      ;FOLD F328 = AUS ;%{SE}%MKUKATPVW %CVW_SPS %VBOASG %P 2:F328 = AUS, 3: BOASG
         $FLAG[328] = FALSE
      ;ENDFOLD
      ;FOLD F324 = AUS ;%{SE}%MKUKATPVW %CVW_SPS %VBOASG %P 2:F324 = AUS, 3: BOASG
         $FLAG[324] = FALSE
      ;ENDFOLD
      ;FOLD Schritt 151 = A4039 ;%{SE}%MKUKATPVW %CVW_SPS %VST_CON %P 2:Schritt 151 = A4039, 3: ST_CON
         IF $OUT[4039] THEN
            PREV_STEP[9] = APP_INT_STEP[9]
            APP_INT_STEP[9] = 151
         ENDIF
      ;ENDFOLD
   ;ENDFOLD
   ;FOLD SCHRITT 151 -- st. RZ1 # Fehler Fraesen -- ;%{P}%MKUKATPVW,%CSTEP,%VST_NR,%P 1:SCHRITT, 2:151, 3: st. RZ1 # Fehler Fraesen
      ;FOLD ;%{H}
         Case 151
      ;ENDFOLD
      ;FOLD -- Fehler Reset AUS -- ;%{SE}%MKUKATPVW %CVW_COM %VCOMMENT %P 2:-- Fehler Reset AUS --, 3: VW_COMMENT
      ;ENDFOLD
      ;FOLD A3857 = AUS ;%{SE}%MKUKATPVW %CVW_SPS %VBOASG %P 2:A3857 = AUS, 3: BOASG
         $OUT[3857] = FALSE
      ;ENDFOLD
      ;FOLD -- Start StartAcknowledge EIN -- ;%{SE}%MKUKATPVW %CVW_COM %VCOMMENT %P 2:-- Start StartAcknowledge EIN --, 3: VW_COMMENT
      ;ENDFOLD
      ;FOLD A3512 = EIN ;%{SE}%MKUKATPVW %CVW_SPS %VBOASG %P 2:A3512 = EIN, 3: BOASG
         $OUT[3512] = TRUE
      ;ENDFOLD
      ;FOLD Schritt 152 = A4039 ;%{SE}%MKUKATPVW %CVW_SPS %VST_CON %P 2:Schritt 152 = A4039, 3: ST_CON
         IF $OUT[4039] THEN
            PREV_STEP[9] = APP_INT_STEP[9]
            APP_INT_STEP[9] = 152
         ENDIF
      ;ENDFOLD
   ;ENDFOLD
   ;FOLD SCHRITT 152 -- st. RZ1 # Fehler Fraesen -- ;%{P}%MKUKATPVW,%CSTEP,%VST_NR,%P 1:SCHRITT, 2:152, 3: st. RZ1 # Fehler Fraesen
      ;FOLD ;%{H}
         Case 152
      ;ENDFOLD
      ;FOLD -- Start StartAcknowledge AUS -- ;%{SE}%MKUKATPVW %CVW_COM %VCOMMENT %P 2:-- Start StartAcknowledge AUS --, 3: VW_COMMENT
      ;ENDFOLD
      ;FOLD A3512 = AUS ;%{SE}%MKUKATPVW %CVW_SPS %VBOASG %P 2:A3512 = AUS, 3: BOASG
         $OUT[3512] = FALSE
      ;ENDFOLD
      ;FOLD -- Start Dress in Position AUS -- ;%{SE}%MKUKATPVW %CVW_COM %VCOMMENT %P 2:-- Start Dress in Position AUS --, 3: VW_COMMENT
      ;ENDFOLD
      ;FOLD A3871 = AUS ;%{SE}%MKUKATPVW %CVW_SPS %VBOASG %P 2:A3871 = AUS, 3: BOASG
         $OUT[3871] = FALSE
      ;ENDFOLD
      ;FOLD -- Start Dress Fin AUS -- ;%{SE}%MKUKATPVW %CVW_COM %VCOMMENT %P 2:-- Start Dress Fin AUS --, 3: VW_COMMENT
      ;ENDFOLD
      ;FOLD A3872 = AUS ;%{SE}%MKUKATPVW %CVW_SPS %VBOASG %P 2:A3872 = AUS, 3: BOASG
         $OUT[3872] = FALSE
      ;ENDFOLD
      ;FOLD -- Start Dress AUS -- ;%{SE}%MKUKATPVW %CVW_COM %VCOMMENT %P 2:-- Start Dress AUS --, 3: VW_COMMENT
      ;ENDFOLD
      ;FOLD A3510 = EIN ;%{SE}%MKUKATPVW %CVW_SPS %VBOASG %P 2:A3510 = EIN, 3: BOASG
         $OUT[3510] = TRUE
      ;ENDFOLD
      ;FOLD -- Start Spot AUS -- ;%{SE}%MKUKATPVW %CVW_COM %VCOMMENT %P 2:-- Start Spot AUS --, 3: VW_COMMENT
      ;ENDFOLD
      ;FOLD A3511 = AUS ;%{SE}%MKUKATPVW %CVW_SPS %VBOASG %P 2:A3511 = AUS, 3: BOASG
         $OUT[3511] = FALSE
      ;ENDFOLD
      ;FOLD -- Start Spot AUS -- ;%{SE}%MKUKATPVW %CVW_COM %VCOMMENT %P 2:-- Start Spot AUS --, 3: VW_COMMENT
      ;ENDFOLD
      ;FOLD A3511 = AUS ;%{SE}%MKUKATPVW %CVW_SPS %VBOASG %P 2:A3511 = AUS, 3: BOASG
         $OUT[3511] = FALSE
      ;ENDFOLD
      ;FOLD -- Start Init Same AUS -- ;%{SE}%MKUKATPVW %CVW_COM %VCOMMENT %P 2:-- Start Init Same AUS --, 3: VW_COMMENT
      ;ENDFOLD
      ;FOLD A3514 = AUS ;%{SE}%MKUKATPVW %CVW_SPS %VBOASG %P 2:A3514 = AUS, 3: BOASG
         $OUT[3514] = FALSE
      ;ENDFOLD
      ;FOLD -- Start Init New AUS -- ;%{SE}%MKUKATPVW %CVW_COM %VCOMMENT %P 2:-- Start Init New AUS --, 3: VW_COMMENT
      ;ENDFOLD
      ;FOLD A3513 = AUS ;%{SE}%MKUKATPVW %CVW_SPS %VBOASG %P 2:A3513 = AUS, 3: BOASG
         $OUT[3513] = FALSE
      ;ENDFOLD
      ;FOLD A3518 = A3519 ;%{SE}%MKUKATPVW %CVW_SPS %VBOASG %P 2:A3518 = A3519, 3: BOASG
         $OUT[3518] = $OUT[3519]
      ;ENDFOLD
      ;FOLD Schritt 153 = A4039 & A3862 ;%{SE}%MKUKATPVW %CVW_SPS %VST_CON %P 2:Schritt 153 = A4039 & A3862, 3: ST_CON
         IF $OUT[4039] AND $OUT[3862] THEN
            PREV_STEP[9] = APP_INT_STEP[9]
            APP_INT_STEP[9] = 153
         ENDIF
      ;ENDFOLD
   ;ENDFOLD
   ;FOLD SCHRITT 153 -- st. RZ1 # Fehler Fraesen -- ;%{P}%MKUKATPVW,%CSTEP,%VST_NR,%P 1:SCHRITT, 2:153, 3: st. RZ1 # Fehler Fraesen
      ;FOLD ;%{H}
         Case 153
      ;ENDFOLD
      ;FOLD -- RSK Fehlerausgabe KF Versetzeinheit -- ;%{SE}%MKUKATPVW %CVW_COM %VCOMMENT %P 2:-- RSK Fehlerausgabe KF Versetzeinheit --, 3: VW_COMMENT
      ;ENDFOLD
      ;FOLD F328 = E835 & F564 ;%{SE}%MKUKATPVW %CVW_SPS %VBOASG %P 2:F328 = E835 & F564, 3: BOASG
         $FLAG[328] = $IN[835] AND $FLAG[564]
      ;ENDFOLD
      ;FOLD -- RSK Fehlerausgabe KS1 Arbeitsstellung -- ;%{SE}%MKUKATPVW %CVW_COM %VCOMMENT %P 2:-- RSK Fehlerausgabe KS1 Arbeitsstellung --, 3: VW_COMMENT
      ;ENDFOLD
      ;FOLD F324 = (E836 + !E837 + !E838 + E839) ;%{SE}%MKUKATPVW %CVW_SPS %VBOASG %P 2:F324 = (E836 + !E837 + !E838 + E839), 3: BOASG
         $FLAG[324] = ($IN[836] OR NOT $IN[837] OR NOT $IN[838] OR $IN[839])
      ;ENDFOLD
      ;FOLD A3519 = EIN ;%{SE}%MKUKATPVW %CVW_SPS %VBOASG %P 2:A3519 = EIN, 3: BOASG
         $OUT[3519] = TRUE
      ;ENDFOLD
      ;FOLD Schritt 154 = A4039 & A3862 & A3505 & A3506 & !A3518 & (E26 + E27) ;%{SE}%MKUKATPVW %CVW_SPS %VST_CON %P 2:Schritt 154 = A4039 & A3862 & A3505 & A3506 & !A3518 & (E26 + E27), 3: ST_CON
         IF $OUT[4039] AND $OUT[3862] AND $OUT[3505] AND $OUT[3506] AND NOT $OUT[3518] AND ($IN[26] OR $IN[27]) THEN
            PREV_STEP[9] = APP_INT_STEP[9]
            APP_INT_STEP[9] = 154
         ENDIF
      ;ENDFOLD
      ;FOLD Schritt 116 = A4039 & A3862 & A3505 & A3506 & A3518 & (E26 + E27) ;%{SE}%MKUKATPVW %CVW_SPS %VST_CON %P 2:Schritt 116 = A4039 & A3862 & A3505 & A3506 & A3518 & (E26 + E27), 3: ST_CON
         IF $OUT[4039] AND $OUT[3862] AND $OUT[3505] AND $OUT[3506] AND $OUT[3518] AND ($IN[26] OR $IN[27]) THEN
            PREV_STEP[9] = APP_INT_STEP[9]
            APP_INT_STEP[9] = 116
         ENDIF
      ;ENDFOLD
   ;ENDFOLD
   ;FOLD SCHRITT 154 -- st. RZ1 # Fehler Fraesen -- ;%{P}%MKUKATPVW,%CSTEP,%VST_NR,%P 1:SCHRITT, 2:154, 3: st. RZ1 # Fehler Fraesen
      ;FOLD ;%{H}
         Case 154
      ;ENDFOLD
      ;FOLD -- Fehler ruecksetzen -- ;%{SE}%MKUKATPVW %CVW_COM %VCOMMENT %P 2:-- Fehler ruecksetzen --, 3: VW_COMMENT
      ;ENDFOLD
      ;FOLD A140 = AUS ;%{SE}%MKUKATPVW %CVW_SPS %VBOASG %P 2:A140 = AUS, 3: BOASG
         $OUT[140] = FALSE
      ;ENDFOLD
      ;FOLD A144 = AUS ;%{SE}%MKUKATPVW %CVW_SPS %VBOASG %P 2:A144 = AUS, 3: BOASG
         $OUT[144] = FALSE
      ;ENDFOLD
      ;FOLD Schritt 103 = (F324 + F328) & E836 & !E837 & !E838 & E839 & A4039 ;%{SE}%MKUKATPVW %CVW_SPS %VST_CON %P 2:Schritt 103 = (F324 + F328) & E836 & !E837 & !E838 & E839 & A4039, 3: ST_CON
         IF ($FLAG[324] OR $FLAG[328]) AND $IN[836] AND NOT $IN[837] AND NOT $IN[838] AND $IN[839] AND $OUT[4039] THEN
            PREV_STEP[9] = APP_INT_STEP[9]
            APP_INT_STEP[9] = 103
         ENDIF
      ;ENDFOLD
      ;FOLD SCHRITT 111 = !F324 & !F328 & !E836 & E837 & E838 & !E839 & A4039 ;%{SE}%MKUKATPVW %CVW_SPS %VST_CON %P 2:SCHRITT 111 = !F324 & !F328 & !E836 & E837 & E838 & !E839 & A4039, 3: ST_CON
         IF NOT $FLAG[324] AND NOT $FLAG[328] AND NOT $IN[836] AND $IN[837] AND $IN[838] AND NOT $IN[839] AND $OUT[4039] THEN
            PREV_STEP[9] = APP_INT_STEP[9]
            APP_INT_STEP[9] = 111
         ENDIF
      ;ENDFOLD
   ;ENDFOLD
   ;FOLD SCHRITT 155 -- st. RZ1 # Fehler Fraesen  -- ;%{P}%MKUKATPVW,%CSTEP,%VST_NR,%P 1:SCHRITT, 2:155, 3: st. RZ1 # Fehler Fraesen
      ;FOLD ;%{H}
         Case 155
      ;ENDFOLD
      ;FOLD Schritt 111 = A4039 & A3506 & A3505 ;%{SE}%MKUKATPVW %CVW_SPS %VST_CON %P 2:Schritt 111 = A4039 & A3506 & A3505, 3: ST_CON
         IF $OUT[4039] AND $OUT[3506] AND $OUT[3505] THEN
            PREV_STEP[9] = APP_INT_STEP[9]
            APP_INT_STEP[9] = 111
         ENDIF
      ;ENDFOLD
   ;ENDFOLD
   ;FOLD SCHRITT 160 -- st. RZ1 # Fehler Messen -- ;%{P}%MKUKATPVW,%CSTEP,%VST_NR,%P 1:SCHRITT, 2:160, 3: st. RZ1 # Fehler Messen
      ;FOLD ;%{H}
         Case 160
      ;ENDFOLD
      ;FOLD 1:;%{SE} %MKUKATPVW
      ;ENDFOLD
   ;ENDFOLD
   ;FOLD SCHRITT 161 -- st. RZ1 # Fehler Messen -- ;%{P}%MKUKATPVW,%CSTEP,%VST_NR,%P 1:SCHRITT, 2:161, 3: st. RZ1 # Fehler Messen
      ;FOLD ;%{H}
         Case 161
      ;ENDFOLD
      ;FOLD -- Fehler Reset AUS -- ;%{SE}%MKUKATPVW %CVW_COM %VCOMMENT %P 2:-- Fehler Reset AUS --, 3: VW_COMMENT
      ;ENDFOLD
      ;FOLD A3857 = AUS ;%{SE}%MKUKATPVW %CVW_SPS %VBOASG %P 2:A3857 = AUS, 3: BOASG
         $OUT[3857] = FALSE
      ;ENDFOLD
      ;FOLD -- Anwahl Zange 1 EIN -- ;%{SE}%MKUKATPVW %CVW_COM %VCOMMENT %P 2:-- Anwahl Zange 1 EIN --, 3: VW_COMMENT
      ;ENDFOLD
      ;FOLD A3858 = EIN ;%{SE}%MKUKATPVW %CVW_SPS %VBOASG %P 2:A3858 = EIN, 3: BOASG
         $OUT[3858] = TRUE
      ;ENDFOLD
      ;FOLD -- Start StartAcknowledge EIN -- ;%{SE}%MKUKATPVW %CVW_COM %VCOMMENT %P 2:-- Start StartAcknowledge EIN --, 3: VW_COMMENT
      ;ENDFOLD
      ;FOLD A3512 = EIN ;%{SE}%MKUKATPVW %CVW_SPS %VBOASG %P 2:A3512 = EIN, 3: BOASG
         $OUT[3512] = TRUE
      ;ENDFOLD
      ;FOLD Schritt 162 = A4039 & A140 & A3862 ;%{SE}%MKUKATPVW %CVW_SPS %VST_CON %P 2:Schritt 162 = A4039 & A140 & A3862, 3: ST_CON
         IF $OUT[4039] AND $OUT[140] AND $OUT[3862] THEN
            PREV_STEP[9] = APP_INT_STEP[9]
            APP_INT_STEP[9] = 162
         ENDIF
      ;ENDFOLD
   ;ENDFOLD
   ;FOLD SCHRITT 162 -- st. RZ1 # Fehler Messen -- ;%{P}%MKUKATPVW,%CSTEP,%VST_NR,%P 1:SCHRITT, 2:162, 3: st. RZ1 # Fehler Messen
      ;FOLD ;%{H}
         Case 162
      ;ENDFOLD
      ;FOLD -- Start Init Same AUS -- ;%{SE}%MKUKATPVW %CVW_COM %VCOMMENT %P 2:-- Start Init Same AUS --, 3: VW_COMMENT
      ;ENDFOLD
      ;FOLD A3514 = AUS ;%{SE}%MKUKATPVW %CVW_SPS %VBOASG %P 2:A3514 = AUS, 3: BOASG
         $OUT[3514] = FALSE
      ;ENDFOLD
      ;FOLD -- Start Spot AUS -- ;%{SE}%MKUKATPVW %CVW_COM %VCOMMENT %P 2:-- Start Spot AUS --, 3: VW_COMMENT
      ;ENDFOLD
      ;FOLD A3511 = AUS ;%{SE}%MKUKATPVW %CVW_SPS %VBOASG %P 2:A3511 = AUS, 3: BOASG
         $OUT[3511] = FALSE
      ;ENDFOLD
      ;FOLD -- Start Dress AUS -- ;%{SE}%MKUKATPVW %CVW_COM %VCOMMENT %P 2:-- Start Dress AUS --, 3: VW_COMMENT
      ;ENDFOLD
      ;FOLD A3510 = AUS ;%{SE}%MKUKATPVW %CVW_SPS %VBOASG %P 2:A3510 = AUS, 3: BOASG
         $OUT[3510] = FALSE
      ;ENDFOLD
      ;FOLD -- Start Init New AUS -- ;%{SE}%MKUKATPVW %CVW_COM %VCOMMENT %P 2:-- Start Init New AUS --, 3: VW_COMMENT
      ;ENDFOLD
      ;FOLD A3513 = AUS ;%{SE}%MKUKATPVW %CVW_SPS %VBOASG %P 2:A3513 = AUS, 3: BOASG
         $OUT[3513] = FALSE
      ;ENDFOLD
      ;FOLD -- Start Dress in Position AUS -- ;%{SE}%MKUKATPVW %CVW_COM %VCOMMENT %P 2:-- Start Dress in Position AUS --, 3: VW_COMMENT
      ;ENDFOLD
      ;FOLD A3871 = AUS ;%{SE}%MKUKATPVW %CVW_SPS %VBOASG %P 2:A3871 = AUS, 3: BOASG
         $OUT[3871] = FALSE
      ;ENDFOLD
      ;FOLD -- Start Dress Fin AUS -- ;%{SE}%MKUKATPVW %CVW_COM %VCOMMENT %P 2:-- Start Dress Fin AUS --, 3: VW_COMMENT
      ;ENDFOLD
      ;FOLD A3872 = AUS ;%{SE}%MKUKATPVW %CVW_SPS %VBOASG %P 2:A3872 = AUS, 3: BOASG
         $OUT[3872] = FALSE
      ;ENDFOLD
      ;FOLD -- Start StartAcknowledge AUS -- ;%{SE}%MKUKATPVW %CVW_COM %VCOMMENT %P 2:-- Start StartAcknowledge AUS --, 3: VW_COMMENT
      ;ENDFOLD
      ;FOLD A3512 = AUS ;%{SE}%MKUKATPVW %CVW_SPS %VBOASG %P 2:A3512 = AUS, 3: BOASG
         $OUT[3512] = FALSE
      ;ENDFOLD
      ;FOLD Schritt 163 = A4039 ;%{SE}%MKUKATPVW %CVW_SPS %VST_CON %P 2:Schritt 163 = A4039, 3: ST_CON
         IF $OUT[4039] THEN
            PREV_STEP[9] = APP_INT_STEP[9]
            APP_INT_STEP[9] = 163
         ENDIF
      ;ENDFOLD
   ;ENDFOLD
   ;FOLD SCHRITT 163 -- st. RZ1 # Fehler Messen -- ;%{P}%MKUKATPVW,%CSTEP,%VST_NR,%P 1:SCHRITT, 2:163, 3: st. RZ1 # Fehler Messen
      ;FOLD ;%{H}
         Case 163
      ;ENDFOLD
      ;FOLD Schritt 164 = A4039 & !A3507 & A3506 & (E26 + E27) ;%{SE}%MKUKATPVW %CVW_SPS %VST_CON %P 2:Schritt 164 = A4039 & !A3507 & A3506 & (E26 + E27), 3: ST_CON
         IF $OUT[4039] AND NOT $OUT[3507] AND $OUT[3506] AND ($IN[26] OR $IN[27]) THEN
            PREV_STEP[9] = APP_INT_STEP[9]
            APP_INT_STEP[9] = 164
         ENDIF
      ;ENDFOLD
   ;ENDFOLD
   ;FOLD SCHRITT 164 -- st. RZ1 # Fehler Messen -- ;%{P}%MKUKATPVW,%CSTEP,%VST_NR,%P 1:SCHRITT, 2:164, 3: st. RZ1 # Fehler Messen
      ;FOLD ;%{H}
         Case 164
      ;ENDFOLD
      ;FOLD Schritt 124 = A4039 & A140 & !A3507 & A3506 & A3505 & F959 ;%{SE}%MKUKATPVW %CVW_SPS %VST_CON %P 2:Schritt 124 = A4039 & A140 & !A3507 & A3506 & A3505 & F959, 3: ST_CON
         IF $OUT[4039] AND $OUT[140] AND NOT $OUT[3507] AND $OUT[3506] AND $OUT[3505] AND $FLAG[959] THEN
            PREV_STEP[9] = APP_INT_STEP[9]
            APP_INT_STEP[9] = 124
         ENDIF
      ;ENDFOLD
   ;ENDFOLD
   ;FOLD SCHRITT 165 --st.RZ1 # Fehler Schweissen-- ;%{P}%MKUKATPVW,%CSTEP,%VST_NR,%P 1:SCHRITT, 2:165, 3:st.RZ1 # Fehler Schweissen
      ;FOLD ;%{H}
         Case 165
      ;ENDFOLD
      ;FOLD -- Start StartAcknowledge AUS -- ;%{SE}%MKUKATPVW %CVW_COM %VCOMMENT %P 2:-- Start StartAcknowledge AUS --, 3: VW_COMMENT
      ;ENDFOLD
      ;FOLD A3512 = AUS ;%{SE}%MKUKATPVW %CVW_SPS %VBOASG %P 2:A3512 = AUS, 3: BOASG
         $OUT[3512] = FALSE
      ;ENDFOLD
      ;FOLD -- Start Dress in Position AUS -- ;%{SE}%MKUKATPVW %CVW_COM %VCOMMENT %P 2:-- Start Dress in Position AUS --, 3: VW_COMMENT
      ;ENDFOLD
      ;FOLD A3871 = AUS ;%{SE}%MKUKATPVW %CVW_SPS %VBOASG %P 2:A3871 = AUS, 3: BOASG
         $OUT[3871] = FALSE
      ;ENDFOLD
      ;FOLD -- Start Dress Fin AUS -- ;%{SE}%MKUKATPVW %CVW_COM %VCOMMENT %P 2:-- Start Dress Fin AUS --, 3: VW_COMMENT
      ;ENDFOLD
      ;FOLD A3872 = AUS ;%{SE}%MKUKATPVW %CVW_SPS %VBOASG %P 2:A3872 = AUS, 3: BOASG
         $OUT[3872] = FALSE
      ;ENDFOLD
      ;FOLD -- Start Dress AUS -- ;%{SE}%MKUKATPVW %CVW_COM %VCOMMENT %P 2:-- Start Dress AUS --, 3: VW_COMMENT
      ;ENDFOLD
      ;FOLD A3510 = AUS ;%{SE}%MKUKATPVW %CVW_SPS %VBOASG %P 2:A3510 = AUS, 3: BOASG
         $OUT[3510] = FALSE
      ;ENDFOLD
      ;FOLD -- Start Spot AUS -- ;%{SE}%MKUKATPVW %CVW_COM %VCOMMENT %P 2:-- Start Spot AUS --, 3: VW_COMMENT
      ;ENDFOLD
      ;FOLD A3511 = AUS ;%{SE}%MKUKATPVW %CVW_SPS %VBOASG %P 2:A3511 = AUS, 3: BOASG
         $OUT[3511] = FALSE
      ;ENDFOLD
      ;FOLD -- Start Spot AUS -- ;%{SE}%MKUKATPVW %CVW_COM %VCOMMENT %P 2:-- Start Spot AUS --, 3: VW_COMMENT
      ;ENDFOLD
      ;FOLD A3511 = AUS ;%{SE}%MKUKATPVW %CVW_SPS %VBOASG %P 2:A3511 = AUS, 3: BOASG
         $OUT[3511] = FALSE
      ;ENDFOLD
      ;FOLD -- Start Init Same AUS -- ;%{SE}%MKUKATPVW %CVW_COM %VCOMMENT %P 2:-- Start Init Same AUS --, 3: VW_COMMENT
      ;ENDFOLD
      ;FOLD A3514 = AUS ;%{SE}%MKUKATPVW %CVW_SPS %VBOASG %P 2:A3514 = AUS, 3: BOASG
         $OUT[3514] = FALSE
      ;ENDFOLD
      ;FOLD -- Start Init New AUS -- ;%{SE}%MKUKATPVW %CVW_COM %VCOMMENT %P 2:-- Start Init New AUS --, 3: VW_COMMENT
      ;ENDFOLD
      ;FOLD A3513 = AUS ;%{SE}%MKUKATPVW %CVW_SPS %VBOASG %P 2:A3513 = AUS, 3: BOASG
         $OUT[3513] = FALSE
      ;ENDFOLD
      ;FOLD A3533 = EIN ;%{SE}%MKUKATPVW %CVW_SPS %VBOASG %P 2:A3533 = EIN, 3: BOASG
         $OUT[3533] = TRUE
      ;ENDFOLD
      ;FOLD A130 = AUS ;%{SE}%MKUKATPVW %CVW_SPS %VBOASG %P 2:A130 = AUS, 3: BOASG
         $OUT[130] = FALSE
      ;ENDFOLD
      ;FOLD F92 = AUS ;%{SE}%MKUKATPVW %CVW_SPS %VBOASG %P 2:F92 = AUS, 3: BOASG
         $FLAG[92] = FALSE
      ;ENDFOLD
      ;FOLD Schritt 2 = A4039 & A3862 & A3506 & A3505 & (E26 + E27) ;%{SE}%MKUKATPVW %CVW_SPS %VST_CON %P 2:Schritt 2 = A4039 & A3862 & A3506 & A3505 & (E26 + E27), 3: ST_CON
         IF $OUT[4039] AND $OUT[3862] AND $OUT[3506] AND $OUT[3505] AND ($IN[26] OR $IN[27]) THEN
            PREV_STEP[9] = APP_INT_STEP[9]
            APP_INT_STEP[9] = 2
         ENDIF
      ;ENDFOLD
   ;ENDFOLD
   ;FOLD SCHRITT 166 --st.RZ1 # Fehler Schweissen-- ;%{P}%MKUKATPVW,%CSTEP,%VST_NR,%P 1:SCHRITT, 2:166, 3:st.RZ1 # Fehler Schweissen
      ;FOLD ;%{H}
         Case 166
      ;ENDFOLD
      ;FOLD 1:;%{SE} %MKUKATPVW
      ;ENDFOLD
   ;ENDFOLD
   ;FOLD SCHRITT 190 -- st. RZ1 Setzhub 2 -- ;%{P}%MKUKATPVW,%CSTEP,%VST_NR,%P 1:SCHRITT, 2:190, 3: st. RZ1 Setzhub 2
      ;FOLD ;%{H}
         Case 190
      ;ENDFOLD
      ;FOLD -- Druckvorgabe SK1/ServoGun -- ;%{SE}%MKUKATPVW %CVW_COM %VCOMMENT %P 2:-- Druckvorgabe SK1/ServoGun --, 3: VW_COMMENT
      ;ENDFOLD
      ;FOLD bin1 ( F78 ) = 61 ;%{SE}%MKUKATPVW %CVW_SPS %VARIASG %P 2:bin1 ( F78 ) = 61, 3: ARIASG
         VW(#BINOUT,$FLAG[78],1,61)
      ;ENDFOLD
      ;FOLD bin31 ( F78 ) = 61 ;%{SE}%MKUKATPVW %CVW_SPS %VARIASG %P 2:bin31 ( F78 ) = 61, 3: ARIASG
         VW(#BINOUT,$FLAG[78],31,61)
      ;ENDFOLD
      ;FOLD -- Wartezeit Programmwechsel SK -- ;%{SE}%MKUKATPVW %CVW_COM %VCOMMENT %P 2:-- Wartezeit Programmwechsel SK --, 3: VW_COMMENT
      ;ENDFOLD
      ;FOLD T8 ( !F334 ) = -2[1/10Sek] ;%{SE}%MKUKATPVW %CVW_SPS %VTASG %P 2:T8 ( !F334 ) = -2[1/10Sek], 3: TASG
         VW(#SET_TIME,NOT $FLAG[334],8,0,-2)
      ;ENDFOLD
      ;FOLD -- Ueberwachungszeit ServoGun Setzhub 2 -- ;%{SE}%MKUKATPVW %CVW_COM %VCOMMENT %P 2:-- Ueberwachungszeit ServoGun Setzhub 2 --, 3: VW_COMMENT
      ;ENDFOLD
      ;FOLD t9 ( EIN ) = -80[1/10Sek] ;%{SE}%MKUKATPVW %CVW_SPS %VTASG %P 2:t9 ( EIN ) = -80[1/10Sek], 3: TASG
         VW(#SET_TIME,TRUE,9,0,-80)
      ;ENDFOLD
      ;FOLD -- Hilfsflag SK Programmwechsel -- ;%{SE}%MKUKATPVW %CVW_COM %VCOMMENT %P 2:-- Hilfsflag SK Programmwechsel --, 3: VW_COMMENT
      ;ENDFOLD
      ;FOLD F334 = EIN ;%{SE}%MKUKATPVW %CVW_SPS %VBOASG %P 2:F334 = EIN, 3: BOASG
         $FLAG[334] = TRUE
      ;ENDFOLD
      ;FOLD A3512 = AUS ;%{SE}%MKUKATPVW %CVW_SPS %VBOASG %P 2:A3512 = AUS, 3: BOASG
         $OUT[3512] = FALSE
      ;ENDFOLD
      ;FOLD SCHRITT 191 = T8 & A4039 & A3506 & A3505 & !A3507 ;%{SE}%MKUKATPVW %CVW_SPS %VST_CON %P 2:SCHRITT 191 = T8 & A4039 & A3506 & A3505 & !A3507, 3: ST_CON
         IF $TIMER_FLAG[8] AND $OUT[4039] AND $OUT[3506] AND $OUT[3505] AND NOT $OUT[3507] THEN
            PREV_STEP[9] = APP_INT_STEP[9]
            APP_INT_STEP[9] = 191
         ENDIF
      ;ENDFOLD
   ;ENDFOLD
   ;FOLD SCHRITT 191 -- st. RZ1 Setzhub 2 # InitSame -- ;%{P}%MKUKATPVW,%CSTEP,%VST_NR,%P 1:SCHRITT, 2:191, 3: st. RZ1 Setzhub 2 # InitSame
      ;FOLD ;%{H}
         Case 191
      ;ENDFOLD
      ;FOLD -- Hilfsflag SK Programmwechsel -- ;%{SE}%MKUKATPVW %CVW_COM %VCOMMENT %P 2:-- Hilfsflag SK Programmwechsel --, 3: VW_COMMENT
      ;ENDFOLD
      ;FOLD F334 = AUS ;%{SE}%MKUKATPVW %CVW_SPS %VBOASG %P 2:F334 = AUS, 3: BOASG
         $FLAG[334] = FALSE
      ;ENDFOLD
      ;FOLD -- Zeit fuer Setzhub -- ;%{SE}%MKUKATPVW %CVW_COM %VCOMMENT %P 2:-- Zeit fuer Setzhub --, 3: VW_COMMENT
      ;ENDFOLD
      ;FOLD T8 ( EIN ) = -80[1/10Sek] ;%{SE}%MKUKATPVW %CVW_SPS %VTASG %P 2:T8 ( EIN ) = -80[1/10Sek], 3: TASG
         VW(#SET_TIME,TRUE,8,0,-80)
      ;ENDFOLD
      ;FOLD -- Messen nach Fraesen -- ;%{SE}%MKUKATPVW %CVW_COM %VCOMMENT %P 2:-- Messen nach Fraesen --, 3: VW_COMMENT
      ;ENDFOLD
      ;FOLD A3514 = EIN ;%{SE}%MKUKATPVW %CVW_SPS %VBOASG %P 2:A3514 = EIN, 3: BOASG
         $OUT[3514] = TRUE
      ;ENDFOLD
      ;FOLD A3510 = EIN ;%{SE}%MKUKATPVW %CVW_SPS %VBOASG %P 2:A3510 = EIN, 3: BOASG
         $OUT[3510] = TRUE
      ;ENDFOLD
      ;FOLD SCHRITT 192 = A4039 ;%{SE}%MKUKATPVW %CVW_SPS %VST_CON %P 2:SCHRITT 192 = A4039, 3: ST_CON
         IF $OUT[4039] THEN
            PREV_STEP[9] = APP_INT_STEP[9]
            APP_INT_STEP[9] = 192
         ENDIF
      ;ENDFOLD
   ;ENDFOLD
   ;FOLD SCHRITT 192 -- st. RZ1 Setzhub 2 # Auswertung -- ;%{P}%MKUKATPVW,%CSTEP,%VST_NR,%P 1:SCHRITT, 2:192, 3: st. RZ1 Setzhub 2 # Auswertung
      ;FOLD ;%{H}
         Case 192
      ;ENDFOLD
      ;FOLD -- Hilfsflag SK Programmwechsel -- ;%{SE}%MKUKATPVW %CVW_COM %VCOMMENT %P 2:-- Hilfsflag SK Programmwechsel --, 3: VW_COMMENT
      ;ENDFOLD
      ;FOLD F334 = AUS ;%{SE}%MKUKATPVW %CVW_SPS %VBOASG %P 2:F334 = AUS, 3: BOASG
         $FLAG[334] = FALSE
      ;ENDFOLD
      ;FOLD -- Warte Ergebnis -- ;%{SE}%MKUKATPVW %CVW_COM %VCOMMENT %P 2:-- Warte Ergebnis --, 3: VW_COMMENT
      ;ENDFOLD
      ;FOLD SCHRITT 193 = A3508 & A4039 + T8 + T9 ;%{SE}%MKUKATPVW %CVW_SPS %VST_CON %P 2:SCHRITT 193 = A3508 & A4039 + T8 + T9, 3: ST_CON
         IF $OUT[3508] AND $OUT[4039] OR $TIMER_FLAG[8] OR $TIMER_FLAG[9] THEN
            PREV_STEP[9] = APP_INT_STEP[9]
            APP_INT_STEP[9] = 193
         ENDIF
      ;ENDFOLD
   ;ENDFOLD
   ;FOLD SCHRITT 193 -- st. RZ1 Setzhub 2 # Acknowledge -- ;%{P}%MKUKATPVW,%CSTEP,%VST_NR,%P 1:SCHRITT, 2:193, 3: st. RZ1 Setzhub 2 # Acknowledge
      ;FOLD ;%{H}
         Case 193
      ;ENDFOLD
      ;FOLD -- RSK Fehlerausgabe Kraftaufbau -- ;%{SE}%MKUKATPVW %CVW_COM %VCOMMENT %P 2:-- RSK Fehlerausgabe Kraftaufbau --, 3: VW_COMMENT
      ;ENDFOLD
      ;FOLD F325 = !A3508 & T9 ;%{SE}%MKUKATPVW %CVW_SPS %VBOASG %P 2:F325 = !A3508 & T9, 3: BOASG
         $FLAG[325] = NOT $OUT[3508] AND $TIMER_FLAG[9]
      ;ENDFOLD
      ;FOLD F329 = T9 ;%{SE}%MKUKATPVW %CVW_SPS %VBOASG %P 2:F329 = T9, 3: BOASG
         $FLAG[329] = $TIMER_FLAG[9]
      ;ENDFOLD
      ;FOLD -- ServoGun SZ1 oeffnen -- ;%{SE}%MKUKATPVW %CVW_COM %VCOMMENT %P 2:-- ServoGun SZ1 oeffnen --, 3: VW_COMMENT
      ;ENDFOLD
      ;FOLD -- RSK Fehlerausgabe Messen -- ;%{SE}%MKUKATPVW %CVW_COM %VCOMMENT %P 2:-- RSK Fehlerausgabe Messen --, 3: VW_COMMENT
      ;ENDFOLD
      ;FOLD A3510 = AUS ;%{SE}%MKUKATPVW %CVW_SPS %VBOASG %P 2:A3510 = AUS, 3: BOASG
         $OUT[3510] = FALSE
      ;ENDFOLD
      ;FOLD A3514 = AUS ;%{SE}%MKUKATPVW %CVW_SPS %VBOASG %P 2:A3514 = AUS, 3: BOASG
         $OUT[3514] = FALSE
      ;ENDFOLD
      ;FOLD A3512 = EIN ;%{SE}%MKUKATPVW %CVW_SPS %VBOASG %P 2:A3512 = EIN, 3: BOASG
         $OUT[3512] = TRUE
      ;ENDFOLD
      ;FOLD -- Druckvorgabe SK1/ServoGun -- ;%{SE}%MKUKATPVW %CVW_COM %VCOMMENT %P 2:-- Druckvorgabe SK1/ServoGun --, 3: VW_COMMENT
      ;ENDFOLD
      ;FOLD bin1 ( F78 ) = 41 ;%{SE}%MKUKATPVW %CVW_SPS %VARIASG %P 2:bin1 ( F78 ) = 41, 3: ARIASG
         VW(#BINOUT,$FLAG[78],1,41)
      ;ENDFOLD
      ;FOLD bin1 ( F79 ) = 51 ;%{SE}%MKUKATPVW %CVW_SPS %VARIASG %P 2:bin1 ( F79 ) = 51, 3: ARIASG
         VW(#BINOUT,$FLAG[79],1,51)
      ;ENDFOLD
      ;FOLD bin31 ( F78 ) = 41 ;%{SE}%MKUKATPVW %CVW_SPS %VARIASG %P 2:bin31 ( F78 ) = 41, 3: ARIASG
         VW(#BINOUT,$FLAG[78],31,41)
      ;ENDFOLD
      ;FOLD bin31 ( F79 ) = 51 ;%{SE}%MKUKATPVW %CVW_SPS %VARIASG %P 2:bin31 ( F79 ) = 51, 3: ARIASG
         VW(#BINOUT,$FLAG[79],31,51)
      ;ENDFOLD
      ;FOLD -- Wartezeit Programmwechsel SK -- ;%{SE}%MKUKATPVW %CVW_COM %VCOMMENT %P 2:-- Wartezeit Programmwechsel SK --, 3: VW_COMMENT
      ;ENDFOLD
      ;FOLD T8 ( !F334 ) = -2[1/10Sek] ;%{SE}%MKUKATPVW %CVW_SPS %VTASG %P 2:T8 ( !F334 ) = -2[1/10Sek], 3: TASG
         VW(#SET_TIME,NOT $FLAG[334],8,0,-2)
      ;ENDFOLD
      ;FOLD -- Hilfsflag SK Programmwechsel -- ;%{SE}%MKUKATPVW %CVW_COM %VCOMMENT %P 2:-- Hilfsflag SK Programmwechsel --, 3: VW_COMMENT
      ;ENDFOLD
      ;FOLD F334 = EIN ;%{SE}%MKUKATPVW %CVW_SPS %VBOASG %P 2:F334 = EIN, 3: BOASG
         $FLAG[334] = TRUE
      ;ENDFOLD
      ;FOLD SCHRITT 194 = T8 & A4039 & !A3507 ;%{SE}%MKUKATPVW %CVW_SPS %VST_CON %P 2:SCHRITT 194 = T8 & A4039 & !A3507, 3: ST_CON
         IF $TIMER_FLAG[8] AND $OUT[4039] AND NOT $OUT[3507] THEN
            PREV_STEP[9] = APP_INT_STEP[9]
            APP_INT_STEP[9] = 194
         ENDIF
      ;ENDFOLD
   ;ENDFOLD
   ;FOLD SCHRITT 194 -- st. RZ1 Setzhub 2 -- ;%{P}%MKUKATPVW,%CSTEP,%VST_NR,%P 1:SCHRITT, 2:194, 3: st. RZ1 Setzhub 2
      ;FOLD ;%{H}
         Case 194
      ;ENDFOLD
      ;FOLD -- Hilfsflag SK Programmwechsel -- ;%{SE}%MKUKATPVW %CVW_COM %VCOMMENT %P 2:-- Hilfsflag SK Programmwechsel --, 3: VW_COMMENT
      ;ENDFOLD
      ;FOLD F334 = AUS ;%{SE}%MKUKATPVW %CVW_SPS %VBOASG %P 2:F334 = AUS, 3: BOASG
         $FLAG[334] = FALSE
      ;ENDFOLD
      ;FOLD A3512 = AUS ;%{SE}%MKUKATPVW %CVW_SPS %VBOASG %P 2:A3512 = AUS, 3: BOASG
         $OUT[3512] = FALSE
      ;ENDFOLD
      ;FOLD SCHRITT 129 = A4039  & A3506 & A3505 & !A3507 ;%{SE}%MKUKATPVW %CVW_SPS %VST_CON %P 2:SCHRITT 129 = A4039  & A3506 & A3505 & !A3507, 3: ST_CON
         IF $OUT[4039] AND $OUT[3506] AND $OUT[3505] AND NOT $OUT[3507] THEN
            PREV_STEP[9] = APP_INT_STEP[9]
            APP_INT_STEP[9] = 129
         ENDIF
      ;ENDFOLD
   ;ENDFOLD
   ;FOLD SCHRITT 203 -- st. RZ2 # Start-- ;%{P}%MKUKATPVW,%CSTEP,%VST_NR,%P 1:SCHRITT, 2:203, 3: st. RZ2 # Start
      ;FOLD ;%{H}
         Case 203
      ;ENDFOLD
      ;FOLD -- RSK gestartet -- ;%{SE}%MKUKATPVW %CVW_COM %VCOMMENT %P 2:-- RSK gestartet --, 3: VW_COMMENT
      ;ENDFOLD
      ;FOLD F160 = AUS ;%{SE}%MKUKATPVW %CVW_SPS %VBOASG %P 2:F160 = AUS, 3: BOASG
         $FLAG[160] = FALSE
      ;ENDFOLD
      ;FOLD F322 = AUS ;%{SE}%MKUKATPVW %CVW_SPS %VBOASG %P 2:F322 = AUS, 3: BOASG
         $FLAG[322] = FALSE
      ;ENDFOLD
      ;FOLD F323 = AUS ;%{SE}%MKUKATPVW %CVW_SPS %VBOASG %P 2:F323 = AUS, 3: BOASG
         $FLAG[323] = FALSE
      ;ENDFOLD
      ;FOLD F324 = AUS ;%{SE}%MKUKATPVW %CVW_SPS %VBOASG %P 2:F324 = AUS, 3: BOASG
         $FLAG[324] = FALSE
      ;ENDFOLD
      ;FOLD F325 = AUS ;%{SE}%MKUKATPVW %CVW_SPS %VBOASG %P 2:F325 = AUS, 3: BOASG
         $FLAG[325] = FALSE
      ;ENDFOLD
      ;FOLD F326 = AUS ;%{SE}%MKUKATPVW %CVW_SPS %VBOASG %P 2:F326 = AUS, 3: BOASG
         $FLAG[326] = FALSE
      ;ENDFOLD
      ;FOLD F327 = AUS ;%{SE}%MKUKATPVW %CVW_SPS %VBOASG %P 2:F327 = AUS, 3: BOASG
         $FLAG[327] = FALSE
      ;ENDFOLD
      ;FOLD F329 = AUS ;%{SE}%MKUKATPVW %CVW_SPS %VBOASG %P 2:F329 = AUS, 3: BOASG
         $FLAG[329] = FALSE
      ;ENDFOLD
      ;FOLD -- ServoGun SZ2 Zaehler -- ;%{SE}%MKUKATPVW %CVW_COM %VCOMMENT %P 2:-- ServoGun SZ2 Zaehler --, 3: VW_COMMENT
      ;ENDFOLD
      ;FOLD F150 = AUS ;%{SE}%MKUKATPVW %CVW_SPS %VBOASG %P 2:F150 = AUS, 3: BOASG
         $FLAG[150] = FALSE
      ;ENDFOLD
      ;FOLD F151 = AUS ;%{SE}%MKUKATPVW %CVW_SPS %VBOASG %P 2:F151 = AUS, 3: BOASG
         $FLAG[151] = FALSE
      ;ENDFOLD
      ;FOLD F152 = AUS ;%{SE}%MKUKATPVW %CVW_SPS %VBOASG %P 2:F152 = AUS, 3: BOASG
         $FLAG[152] = FALSE
      ;ENDFOLD
      ;FOLD F153 = AUS ;%{SE}%MKUKATPVW %CVW_SPS %VBOASG %P 2:F153 = AUS, 3: BOASG
         $FLAG[153] = FALSE
      ;ENDFOLD
      ;FOLD F154 = AUS ;%{SE}%MKUKATPVW %CVW_SPS %VBOASG %P 2:F154 = AUS, 3: BOASG
         $FLAG[154] = FALSE
      ;ENDFOLD
      ;FOLD F155 = AUS ;%{SE}%MKUKATPVW %CVW_SPS %VBOASG %P 2:F155 = AUS, 3: BOASG
         $FLAG[155] = FALSE
      ;ENDFOLD
      ;FOLD -- Hilfsflags Funktionstest KF Motor -- ;%{SE}%MKUKATPVW %CVW_COM %VCOMMENT %P 2:-- Hilfsflags Funktionstest KF Motor --, 3: VW_COMMENT
      ;ENDFOLD
      ;FOLD F312 = AUS ;%{SE}%MKUKATPVW %CVW_SPS %VBOASG %P 2:F312 = AUS, 3: BOASG
         $FLAG[312] = FALSE
      ;ENDFOLD
      ;FOLD F313 = AUS ;%{SE}%MKUKATPVW %CVW_SPS %VBOASG %P 2:F313 = AUS, 3: BOASG
         $FLAG[313] = FALSE
      ;ENDFOLD
      ;FOLD -- Hilfsflags ServoGun Start -- ;%{SE}%MKUKATPVW %CVW_COM %VCOMMENT %P 2:-- Hilfsflags ServoGun Start --, 3: VW_COMMENT
      ;ENDFOLD
      ;FOLD F276 = EIN ;%{SE}%MKUKATPVW %CVW_SPS %VBOASG %P 2:F276 = EIN, 3: BOASG
         $FLAG[276] = TRUE
      ;ENDFOLD
      ;FOLD A3903 = AUS ;%{SE}%MKUKATPVW %CVW_SPS %VBOASG %P 2:A3903 = AUS, 3: BOASG
         $OUT[3903] = FALSE
      ;ENDFOLD
      ;FOLD A3904 = AUS ;%{SE}%MKUKATPVW %CVW_SPS %VBOASG %P 2:A3904 = AUS, 3: BOASG
         $OUT[3904] = FALSE
      ;ENDFOLD
      ;FOLD A3510 = EIN ;%{SE}%MKUKATPVW %CVW_SPS %VBOASG %P 2:A3510 = EIN, 3: BOASG
         $OUT[3510] = TRUE
      ;ENDFOLD
      ;FOLD A3511 = AUS ;%{SE}%MKUKATPVW %CVW_SPS %VBOASG %P 2:A3511 = AUS, 3: BOASG
         $OUT[3511] = FALSE
      ;ENDFOLD
      ;FOLD A3514 = AUS ;%{SE}%MKUKATPVW %CVW_SPS %VBOASG %P 2:A3514 = AUS, 3: BOASG
         $OUT[3514] = FALSE
      ;ENDFOLD
      ;FOLD A3513 = AUS ;%{SE}%MKUKATPVW %CVW_SPS %VBOASG %P 2:A3513 = AUS, 3: BOASG
         $OUT[3513] = FALSE
      ;ENDFOLD
      ;FOLD A3512 = AUS ;%{SE}%MKUKATPVW %CVW_SPS %VBOASG %P 2:A3512 = AUS, 3: BOASG
         $OUT[3512] = FALSE
      ;ENDFOLD
      ;FOLD A3534 = AUS ;%{SE}%MKUKATPVW %CVW_SPS %VBOASG %P 2:A3534 = AUS, 3: BOASG
         $OUT[3534] = FALSE
      ;ENDFOLD
      ;FOLD A3535 = AUS ;%{SE}%MKUKATPVW %CVW_SPS %VBOASG %P 2:A3535 = AUS, 3: BOASG
         $OUT[3535] = FALSE
      ;ENDFOLD
      ;FOLD A3536 = AUS ;%{SE}%MKUKATPVW %CVW_SPS %VBOASG %P 2:A3536 = AUS, 3: BOASG
         $OUT[3536] = FALSE
      ;ENDFOLD
      ;FOLD -- Hilfsflags ServoGun Ende -- ;%{SE}%MKUKATPVW %CVW_COM %VCOMMENT %P 2:-- Hilfsflags ServoGun Ende --, 3: VW_COMMENT
      ;ENDFOLD
      ;FOLD -- Ausblasen zuruecksetzen -- ;%{SE}%MKUKATPVW %CVW_COM %VCOMMENT %P 2:-- Ausblasen zuruecksetzen --, 3: VW_COMMENT
      ;ENDFOLD
      ;FOLD A836 = AUS ;%{SE}%MKUKATPVW %CVW_SPS %VBOASG %P 2:A836 = AUS, 3: BOASG
         $OUT[836] = FALSE
      ;ENDFOLD
      ;FOLD A996 = AUS ;%{SE}%MKUKATPVW %CVW_SPS %VBOASG %P 2:A996 = AUS, 3: BOASG
         $OUT[996] = FALSE
      ;ENDFOLD
      ;FOLD A1156 = AUS ;%{SE}%MKUKATPVW %CVW_SPS %VBOASG %P 2:A1156 = AUS, 3: BOASG
         $OUT[1156] = FALSE
      ;ENDFOLD
      ;FOLD -- Prognummer setzen -- ;%{SE}%MKUKATPVW %CVW_COM %VCOMMENT %P 2:-- Prognummer setzen --, 3: VW_COMMENT
      ;ENDFOLD
      ;FOLD bin28 ( EIN ) = 0 ;%{SE}%MKUKATPVW %CVW_SPS %VARIASG %P 2:bin28 ( EIN ) = 0, 3: ARIASG
         VW(#BINOUT,TRUE,28,0)
      ;ENDFOLD
      ;FOLD bin6 ( EIN ) = 31 ;%{SE}%MKUKATPVW %CVW_SPS %VARIASG %P 2:bin6 ( EIN ) = 31, 3: ARIASG
         VW(#BINOUT,TRUE,6,31)
      ;ENDFOLD
      ;FOLD bin30 ( EIN ) = p112 ;%{SE}%MKUKATPVW %CVW_SPS %VARIASG %P 2:bin30 ( EIN ) = p112, 3: ARIASG
         VW(#BINOUT,TRUE,30,PROCPAR[112])
      ;ENDFOLD
      ;FOLD bin31 ( EIN ) = 31 ;%{SE}%MKUKATPVW %CVW_SPS %VARIASG %P 2:bin31 ( EIN ) = 31, 3: ARIASG
         VW(#BINOUT,TRUE,31,31)
      ;ENDFOLD
      ;FOLD -- Wartezeit Programmwechsel SK -- ;%{SE}%MKUKATPVW %CVW_COM %VCOMMENT %P 2:-- Wartezeit Programmwechsel SK --, 3: VW_COMMENT
      ;ENDFOLD
      ;FOLD T8 ( !F334 ) = -2[1/10Sek] ;%{SE}%MKUKATPVW %CVW_SPS %VTASG %P 2:T8 ( !F334 ) = -2[1/10Sek], 3: TASG
         VW(#SET_TIME,NOT $FLAG[334],8,0,-2)
      ;ENDFOLD
      ;FOLD -- Hilfsflag SK Programmwechsel -- ;%{SE}%MKUKATPVW %CVW_COM %VCOMMENT %P 2:-- Hilfsflag SK Programmwechsel --, 3: VW_COMMENT
      ;ENDFOLD
      ;FOLD F334 = EIN ;%{SE}%MKUKATPVW %CVW_SPS %VBOASG %P 2:F334 = EIN, 3: BOASG
         $FLAG[334] = TRUE
      ;ENDFOLD
      ;FOLD -- Stat. ServoGun SZ1 beim Fraesen -- ;%{SE}%MKUKATPVW %CVW_COM %VCOMMENT %P 2:-- Stat. ServoGun SZ1 beim Fraesen --, 3: VW_COMMENT
      ;ENDFOLD
      ;FOLD A116 = EIN ;%{SE}%MKUKATPVW %CVW_SPS %VBOASG %P 2:A116 = EIN, 3: BOASG
         $OUT[116] = TRUE
      ;ENDFOLD
      ;FOLD A162 = EIN ;%{SE}%MKUKATPVW %CVW_SPS %VBOASG %P 2:A162 = EIN, 3: BOASG
         $OUT[162] = TRUE
      ;ENDFOLD
      ;FOLD -- Schritt Fraesen aktiv -- ;%{SE}%MKUKATPVW %CVW_COM %VCOMMENT %P 2:-- Schritt Fraesen aktiv --, 3: VW_COMMENT
      ;ENDFOLD
      ;FOLD A3534 = EIN ;%{SE}%MKUKATPVW %CVW_SPS %VBOASG %P 2:A3534 = EIN, 3: BOASG
         $OUT[3534] = TRUE
      ;ENDFOLD
      ;FOLD -- Quitt. Fraesen SK1 AUS -- ;%{SE}%MKUKATPVW %CVW_COM %VCOMMENT %P 2:-- Quitt. Fraesen SK1 AUS --, 3: VW_COMMENT
      ;ENDFOLD
      ;FOLD A946 = F830 ;%{SE}%MKUKATPVW %CVW_SPS %VBOASG %P 2:A946 = F830, 3: BOASG
         $OUT[946] = $FLAG[830]
      ;ENDFOLD
      ;FOLD A882 = !F830 ;%{SE}%MKUKATPVW %CVW_SPS %VBOASG %P 2:A882 = !F830, 3: BOASG
         $OUT[882] = NOT $FLAG[830]
      ;ENDFOLD
      ;FOLD SCHRITT 204 = A4039 ;%{SE}%MKUKATPVW %CVW_SPS %VST_CON %P 2:SCHRITT 204 = A4039, 3: ST_CON
         IF $OUT[4039] THEN
            PREV_STEP[9] = APP_INT_STEP[9]
            APP_INT_STEP[9] = 204
         ENDIF
      ;ENDFOLD
   ;ENDFOLD
   ;FOLD SCHRITT 204 -- st. RZ2 -- ;%{P}%MKUKATPVW,%CSTEP,%VST_NR,%P 1:SCHRITT, 2:204, 3: st. RZ2
      ;FOLD ;%{H}
         Case 204
      ;ENDFOLD
      ;FOLD -- Hilfsflag SK Programmwechsel -- ;%{SE}%MKUKATPVW %CVW_COM %VCOMMENT %P 2:-- Hilfsflag SK Programmwechsel --, 3: VW_COMMENT
      ;ENDFOLD
      ;FOLD F334 = AUS ;%{SE}%MKUKATPVW %CVW_SPS %VBOASG %P 2:F334 = AUS, 3: BOASG
         $FLAG[334] = FALSE
      ;ENDFOLD
      ;FOLD -- Wiederholfraesen aktiv -- ;%{SE}%MKUKATPVW %CVW_COM %VCOMMENT %P 2:-- Wiederholfraesen aktiv --, 3: VW_COMMENT
      ;ENDFOLD
      ;FOLD F327 = A3519 ;%{SE}%MKUKATPVW %CVW_SPS %VBOASG %P 2:F327 = A3519, 3: BOASG
         $FLAG[327] = $OUT[3519]
      ;ENDFOLD
      ;FOLD F749 = A3519 ;%{SE}%MKUKATPVW %CVW_SPS %VBOASG %P 2:F749 = A3519, 3: BOASG
         $FLAG[749] = $OUT[3519]
      ;ENDFOLD
      ;FOLD A176 = AUS ;%{SE}%MKUKATPVW %CVW_SPS %VBOASG %P 2:A176 = AUS, 3: BOASG
         $OUT[176] = FALSE
      ;ENDFOLD
      ;FOLD -- Ueberwachungszeit KF1 EIN -- ;%{SE}%MKUKATPVW %CVW_COM %VCOMMENT %P 2:-- Ueberwachungszeit KF1 EIN --, 3: VW_COMMENT
      ;ENDFOLD
      ;FOLD T7 ( EIN ) = -50[1/10Sek] ;%{SE}%MKUKATPVW %CVW_SPS %VTASG %P 2:T7 ( EIN ) = -50[1/10Sek], 3: TASG
         VW(#SET_TIME,TRUE,7,0,-50)
      ;ENDFOLD
      ;FOLD -- KF1 einschalten -- ;%{SE}%MKUKATPVW %CVW_COM %VCOMMENT %P 2:-- KF1 einschalten --, 3: VW_COMMENT
      ;ENDFOLD
      ;FOLD i1 (EIN) = 0 ;%{SE}%MKUKATPVW %CVW_SPS %VARIASG %P 2:i1 (EIN) = 0, 3: ARIASG
         VW(#COUNTER,TRUE,1,0)
      ;ENDFOLD
      ;FOLD A994 = EIN ;%{SE}%MKUKATPVW %CVW_SPS %VBOASG %P 2:A994 = EIN, 3: BOASG
         $OUT[994] = TRUE
      ;ENDFOLD
      ;FOLD SCHRITT 205 = A4039 ;%{SE}%MKUKATPVW %CVW_SPS %VST_CON %P 2:SCHRITT 205 = A4039, 3: ST_CON
         IF $OUT[4039] THEN
            PREV_STEP[9] = APP_INT_STEP[9]
            APP_INT_STEP[9] = 205
         ENDIF
      ;ENDFOLD
   ;ENDFOLD
   ;FOLD SCHRITT 205 -- st. RZ2 # Funktionstest KF -- ;%{P}%MKUKATPVW,%CSTEP,%VST_NR,%P 1:SCHRITT, 2:205, 3: st. RZ2 # Funktionstest KF
      ;FOLD ;%{H}
         Case 205
      ;ENDFOLD
      ;FOLD -- Funktionstest KF Motor -- ;%{SE}%MKUKATPVW %CVW_COM %VCOMMENT %P 2:-- Funktionstest KF Motor --, 3: VW_COMMENT
      ;ENDFOLD
      ;FOLD F312 = EIN ;%{SE}%MKUKATPVW %CVW_SPS %VBOASG %P 2:F312 = EIN, 3: BOASG
         $FLAG[312] = TRUE
      ;ENDFOLD
      ;FOLD F313 = i1 > 2 ;%{SE}%MKUKATPVW %CVW_SPS %VBOCMP %P 2:F313 = i1 > 2, 3: BOCMP
         $FLAG[313] = $COUNT_I[1] > 2
      ;ENDFOLD
      ;FOLD -- Ueberwachungszeit KS1 schwenken -- ;%{SE}%MKUKATPVW %CVW_COM %VCOMMENT %P 2:-- Ueberwachungszeit KS1 schwenken --, 3: VW_COMMENT
      ;ENDFOLD
      ;FOLD t8 ( EIN ) = -100[1/10Sek] ;%{SE}%MKUKATPVW %CVW_SPS %VTASG %P 2:t8 ( EIN ) = -100[1/10Sek], 3: TASG
         VW(#SET_TIME,TRUE,8,0,-100)
      ;ENDFOLD
      ;FOLD Schritt 207 = (F313 + T7) & A4039 ;%{SE}%MKUKATPVW %CVW_SPS %VST_CON %P 2:Schritt 207 = (F313 + T7) & A4039, 3: ST_CON
         IF ($FLAG[313] OR $TIMER_FLAG[7]) AND $OUT[4039] THEN
            PREV_STEP[9] = APP_INT_STEP[9]
            APP_INT_STEP[9] = 207
         ENDIF
      ;ENDFOLD
   ;ENDFOLD
   ;FOLD SCHRITT 207 -- st. RZ2 # Fehler KF -- ;%{P}%MKUKATPVW,%CSTEP,%VST_NR,%P 1:SCHRITT, 2:207, 3: st. RZ2 # Fehler KF
      ;FOLD ;%{H}
         Case 207
      ;ENDFOLD
      ;FOLD -- RSK Fehlerausgabe KF1 Initiator/Motor -- ;%{SE}%MKUKATPVW %CVW_COM %VCOMMENT %P 2:-- RSK Fehlerausgabe KF1 Initiator/Motor --, 3: VW_COMMENT
      ;ENDFOLD
      ;FOLD F322 = !F313 ;%{SE}%MKUKATPVW %CVW_SPS %VBOASG %P 2:F322 = !F313, 3: BOASG
         $FLAG[322] = NOT $FLAG[313]
      ;ENDFOLD
      ;FOLD -- RSK Fehlerausgabe KS1 Ruhest. -- ;%{SE}%MKUKATPVW %CVW_COM %VCOMMENT %P 2:-- RSK Fehlerausgabe KS1 Ruhest. --, 3: VW_COMMENT
      ;ENDFOLD
      ;FOLD F323 = (!E996 + E997 + E998 + !E999) & !F324 & !F328 ;%{SE}%MKUKATPVW %CVW_SPS %VBOASG %P 2:F323 = (!E996 + E997 + E998 + !E999) & !F324 & !F328, 3: BOASG
         $FLAG[323] = (NOT $IN[996] OR $IN[997] OR $IN[998] OR NOT $IN[999]) AND NOT $FLAG[324] AND NOT $FLAG[328]
      ;ENDFOLD
      ;FOLD -- RSK Sammelstoerung -- ;%{SE}%MKUKATPVW %CVW_COM %VCOMMENT %P 2:-- RSK Sammelstoerung --, 3: VW_COMMENT
      ;ENDFOLD
      ;FOLD F329 = F322 + F323 + T8 ;%{SE}%MKUKATPVW %CVW_SPS %VBOASG %P 2:F329 = F322 + F323 + T8, 3: BOASG
         $FLAG[329] = $FLAG[322] OR $FLAG[323] OR $TIMER_FLAG[8]
      ;ENDFOLD
      ;FOLD T7 ( EIN ) = STOP ;%{SE}%MKUKATPVW %CVW_SPS %VTSTOP %P 2:T7 ( EIN ) = STOP, 3: TSTOP
         VW(#SET_TIME,TRUE,7,1,0)
      ;ENDFOLD
      ;FOLD -- KF Motor Ein -- ;%{SE}%MKUKATPVW %CVW_COM %VCOMMENT %P 2:-- KF Motor Ein --, 3: VW_COMMENT
      ;ENDFOLD
      ;FOLD A994 = !F322 & !F323 ;%{SE}%MKUKATPVW %CVW_SPS %VBOASG %P 2:A994 = !F322 & !F323, 3: BOASG
         $OUT[994] = NOT $FLAG[322] AND NOT $FLAG[323]
      ;ENDFOLD
      ;FOLD -- KF1 Versetzeinheit vor -- ;%{SE}%MKUKATPVW %CVW_COM %VCOMMENT %P 2:-- KF1 Versetzeinheit vor --, 3: VW_COMMENT
      ;ENDFOLD
      ;FOLD A995 = !F322 & !F323 & F564 ;%{SE}%MKUKATPVW %CVW_SPS %VBOASG %P 2:A995 = !F322 & !F323 & F564, 3: BOASG
         $OUT[995] = NOT $FLAG[322] AND NOT $FLAG[323] AND $FLAG[564]
      ;ENDFOLD
      ;FOLD SCHRITT 208 = (!F322 & !F323) & (E995 & F564 + !E995 & !F564) & A4039 ;%{SE}%MKUKATPVW %CVW_SPS %VST_CON %P 2:SCHRITT 208 = (!F322 & !F323) & (E995 & F564 + !E995 & !F564) & A4039, 3: ST_CON
         IF (NOT $FLAG[322] AND NOT $FLAG[323]) AND ($IN[995] AND $FLAG[564] OR NOT $IN[995] AND NOT $FLAG[564]) AND $OUT[4039] THEN
            PREV_STEP[9] = APP_INT_STEP[9]
            APP_INT_STEP[9] = 208
         ENDIF
      ;ENDFOLD
      ;FOLD SCHRITT 234 = (F322 + F323) & !F324 & !F328 & A4039 & (E26 + E27) ;%{SE}%MKUKATPVW %CVW_SPS %VST_CON %P 2:SCHRITT 234 = (F322 + F323) & !F324 & !F328 & A4039 & (E26 + E27), 3: ST_CON
         IF ($FLAG[322] OR $FLAG[323]) AND NOT $FLAG[324] AND NOT $FLAG[328] AND $OUT[4039] AND ($IN[26] OR $IN[27]) THEN
            PREV_STEP[9] = APP_INT_STEP[9]
            APP_INT_STEP[9] = 234
         ENDIF
      ;ENDFOLD
   ;ENDFOLD
   ;FOLD SCHRITT 208 -- st. RZ2 # Sicherheit KF -- ;%{P}%MKUKATPVW,%CSTEP,%VST_NR,%P 1:SCHRITT, 2:208, 3: st. RZ2 # Sicherheit KF
      ;FOLD ;%{H}
         Case 208
      ;ENDFOLD
      ;FOLD -- RSK Sammelstoerung -- ;%{SE}%MKUKATPVW %CVW_COM %VCOMMENT %P 2:-- RSK Sammelstoerung --, 3: VW_COMMENT
      ;ENDFOLD
      ;FOLD F329 = AUS ;%{SE}%MKUKATPVW %CVW_SPS %VBOASG %P 2:F329 = AUS, 3: BOASG
         $FLAG[329] = FALSE
      ;ENDFOLD
      ;FOLD F324 = AUS ;%{SE}%MKUKATPVW %CVW_SPS %VBOASG %P 2:F324 = AUS, 3: BOASG
         $FLAG[324] = FALSE
      ;ENDFOLD
      ;FOLD F328 = AUS ;%{SE}%MKUKATPVW %CVW_SPS %VBOASG %P 2:F328 = AUS, 3: BOASG
         $FLAG[328] = FALSE
      ;ENDFOLD
      ;FOLD -- Wartebedingung schwenken -- ;%{SE}%MKUKATPVW %CVW_COM %VCOMMENT %P 2:-- Wartebedingung schwenken --, 3: VW_COMMENT
      ;ENDFOLD
      ;FOLD Schritt 209 = A3894 & A4039 ;%{SE}%MKUKATPVW %CVW_SPS %VST_CON %P 2:Schritt 209 = A3894 & A4039, 3: ST_CON
         IF $OUT[3894] AND $OUT[4039] THEN
            PREV_STEP[9] = APP_INT_STEP[9]
            APP_INT_STEP[9] = 209
         ENDIF
      ;ENDFOLD
   ;ENDFOLD
   ;FOLD SCHRITT 209 -- st. RZ2 # KS in AS schwenken -- ;%{P}%MKUKATPVW,%CSTEP,%VST_NR,%P 1:SCHRITT, 2:209, 3: st. RZ2 # KS in AS schwenken
      ;FOLD ;%{H}
         Case 209
      ;ENDFOLD
      ;FOLD -- KS1 in Arbeitsstellung schwenken -- ;%{SE}%MKUKATPVW %CVW_COM %VCOMMENT %P 2:-- KS1 in Arbeitsstellung schwenken --, 3: VW_COMMENT
      ;ENDFOLD
      ;FOLD A1000 = A3894 & !E997 & (E995 & F564 + !E995 & !F564) ;%{SE}%MKUKATPVW %CVW_SPS %VBOASG %P 2:A1000 = A3894 & !E997 & (E995 & F564 + !E995 & !F564), 3: BOASG
         $OUT[1000] = $OUT[3894] AND NOT $IN[997] AND ($IN[995] AND $FLAG[564] OR NOT $IN[995] AND NOT $FLAG[564])
      ;ENDFOLD
      ;FOLD -- KF1 Ausblasen -- ;%{SE}%MKUKATPVW %CVW_COM %VCOMMENT %P 2:-- KF1 Ausblasen --, 3: VW_COMMENT
      ;ENDFOLD
      ;FOLD A996 = F330 + !F330 & !F331 & !F332 ;%{SE}%MKUKATPVW %CVW_SPS %VBOASG %P 2:A996 = F330 + !F330 & !F331 & !F332, 3: BOASG
         $OUT[996] = $FLAG[330] OR NOT $FLAG[330] AND NOT $FLAG[331] AND NOT $FLAG[332]
      ;ENDFOLD
      ;FOLD Schritt 210 = A3894 & (A1000 + E997 + T8) & A4039 ;%{SE}%MKUKATPVW %CVW_SPS %VST_CON %P 2:Schritt 210 = A3894 & (A1000 + E997 + T8) & A4039, 3: ST_CON
         IF $OUT[3894] AND ($OUT[1000] OR $IN[997] OR $TIMER_FLAG[8]) AND $OUT[4039] THEN
            PREV_STEP[9] = APP_INT_STEP[9]
            APP_INT_STEP[9] = 210
         ENDIF
      ;ENDFOLD
   ;ENDFOLD
   ;FOLD SCHRITT 210 -- st. RZ2 -- ;%{P}%MKUKATPVW,%CSTEP,%VST_NR,%P 1:SCHRITT, 2:210, 3: st. RZ2
      ;FOLD ;%{H}
         Case 210
      ;ENDFOLD
      ;FOLD -- RSK Fehlerausgabe KF Versetzeinheit -- ;%{SE}%MKUKATPVW %CVW_COM %VCOMMENT %P 2:-- RSK Fehlerausgabe KF Versetzeinheit --, 3: VW_COMMENT
      ;ENDFOLD
      ;FOLD F328 = !E995 & F564 & !F324 ;%{SE}%MKUKATPVW %CVW_SPS %VBOASG %P 2:F328 = !E995 & F564 & !F324, 3: BOASG
         $FLAG[328] = NOT $IN[995] AND $FLAG[564] AND NOT $FLAG[324]
      ;ENDFOLD
      ;FOLD -- RSK Fehlerausgabe KS1 Arbeitsstellung -- ;%{SE}%MKUKATPVW %CVW_COM %VCOMMENT %P 2:-- RSK Fehlerausgabe KS1 Arbeitsstellung --, 3: VW_COMMENT
      ;ENDFOLD
      ;FOLD F324 = (E996 + !E997 + !E998 + E999) & T8 & (E995 + !F564) + F324 ;%{SE}%MKUKATPVW %CVW_SPS %VBOASG %P 2:F324 = (E996 + !E997 + !E998 + E999) & T8 & (E995 + !F564) + F324, 3: BOASG
         $FLAG[324] = ($IN[996] OR NOT $IN[997] OR NOT $IN[998] OR $IN[999]) AND $TIMER_FLAG[8] AND ($IN[995] OR NOT $FLAG[564]) OR $FLAG[324]
      ;ENDFOLD
      ;FOLD -- RSK Fehlerausgabe EZ/SP min. Oeffnung -- ;%{SE}%MKUKATPVW %CVW_COM %VCOMMENT %P 2:-- RSK Fehlerausgabe EZ/SP min. Oeffnung --, 3: VW_COMMENT
      ;ENDFOLD
      ;FOLD F333 = !A3894 ;%{SE}%MKUKATPVW %CVW_SPS %VBOASG %P 2:F333 = !A3894, 3: BOASG
         $FLAG[333] = NOT $OUT[3894]
      ;ENDFOLD
      ;FOLD -- RSK Sammelstoerung -- ;%{SE}%MKUKATPVW %CVW_COM %VCOMMENT %P 2:-- RSK Sammelstoerung --, 3: VW_COMMENT
      ;ENDFOLD
      ;FOLD F329 = F324 + F328 + F333 ;%{SE}%MKUKATPVW %CVW_SPS %VBOASG %P 2:F329 = F324 + F328 + F333, 3: BOASG
         $FLAG[329] = $FLAG[324] OR $FLAG[328] OR $FLAG[333]
      ;ENDFOLD
      ;FOLD A994 = !F324 & !F328 ;%{SE}%MKUKATPVW %CVW_SPS %VBOASG %P 2:A994 = !F324 & !F328, 3: BOASG
         $OUT[994] = NOT $FLAG[324] AND NOT $FLAG[328]
      ;ENDFOLD
      ;FOLD -- KF1 Ausblasen -- ;%{SE}%MKUKATPVW %CVW_COM %VCOMMENT %P 2:-- KF1 Ausblasen --, 3: VW_COMMENT
      ;ENDFOLD
      ;FOLD A996 = (F330 + !F330 & !F331 & !F332) & !F324 & !F328 ;%{SE}%MKUKATPVW %CVW_SPS %VBOASG %P 2:A996 = (F330 + !F330 & !F331 & !F332) & !F324 & !F328, 3: BOASG
         $OUT[996] = ($FLAG[330] OR NOT $FLAG[330] AND NOT $FLAG[331] AND NOT $FLAG[332]) AND NOT $FLAG[324] AND NOT $FLAG[328]
      ;ENDFOLD
      ;FOLD A995 = F564 ;%{SE}%MKUKATPVW %CVW_SPS %VBOASG %P 2:A995 = F564, 3: BOASG
         $OUT[995] = $FLAG[564]
      ;ENDFOLD
      ;FOLD -- Verweilzeit Versetzeinheit Rueck -- ;%{SE}%MKUKATPVW %CVW_COM %VCOMMENT %P 2:-- Verweilzeit Versetzeinheit Rueck --, 3: VW_COMMENT
      ;ENDFOLD
      ;FOLD t11 ( EIN ) = i24[1/10Sek] ;%{SE}%MKUKATPVW %CVW_SPS %VTASG %P 2:t11 ( EIN ) = i24[1/10Sek], 3: TASG
         VW(#SET_TIME,TRUE,11,0,$COUNT_I[24])
      ;ENDFOLD
      ;FOLD SCHRITT 203 = (F324 + F328) & (E26 + E27) & A4039 ;%{SE}%MKUKATPVW %CVW_SPS %VST_CON %P 2:SCHRITT 203 = (F324 + F328) & (E26 + E27) & A4039, 3: ST_CON
         IF ($FLAG[324] OR $FLAG[328]) AND ($IN[26] OR $IN[27]) AND $OUT[4039] THEN
            PREV_STEP[9] = APP_INT_STEP[9]
            APP_INT_STEP[9] = 203
         ENDIF
      ;ENDFOLD
      ;FOLD SCHRITT 211 = !F324 & !F328 & !E996 & E997 & E998 & !E999 & A4039 ;%{SE}%MKUKATPVW %CVW_SPS %VST_CON %P 2:SCHRITT 211 = !F324 & !F328 & !E996 & E997 & E998 & !E999 & A4039, 3: ST_CON
         IF NOT $FLAG[324] AND NOT $FLAG[328] AND NOT $IN[996] AND $IN[997] AND $IN[998] AND NOT $IN[999] AND $OUT[4039] THEN
            PREV_STEP[9] = APP_INT_STEP[9]
            APP_INT_STEP[9] = 211
         ENDIF
      ;ENDFOLD
   ;ENDFOLD
   ;FOLD SCHRITT 211 -- st. RZ2 -- ;%{P}%MKUKATPVW,%CSTEP,%VST_NR,%P 1:SCHRITT, 2:211, 3: st. RZ2
      ;FOLD ;%{H}
         Case 211
      ;ENDFOLD
      ;FOLD -- Umdreh. KF setzen zwischenspeichern -- ;%{SE}%MKUKATPVW %CVW_COM %VCOMMENT %P 2:-- Umdreh. KF setzen zwischenspeichern --, 3: VW_COMMENT
      ;ENDFOLD
      ;FOLD i45 ( EIN ) = i7 ;%{SE}%MKUKATPVW %CVW_SPS %VARIASG %P 2:i45 ( EIN ) = i7, 3: ARIASG
         VW(#COUNTER,TRUE,45,$COUNT_I[7])
      ;ENDFOLD
      ;FOLD i7 ( F155 ) = i43 ;%{SE}%MKUKATPVW %CVW_SPS %VARIASG %P 2:i7 ( F155 ) = i43, 3: ARIASG
         VW(#COUNTER,$FLAG[155],7,$COUNT_I[43])
      ;ENDFOLD
      ;FOLD i1 ( EIN ) = 0 ;%{SE}%MKUKATPVW %CVW_SPS %VARIASG %P 2:i1 ( EIN ) = 0, 3: ARIASG
         VW(#COUNTER,TRUE,1,0)
      ;ENDFOLD
      ;FOLD F154 = AUS ;%{SE}%MKUKATPVW %CVW_SPS %VBOASG %P 2:F154 = AUS, 3: BOASG
         $FLAG[154] = FALSE
      ;ENDFOLD
      ;FOLD F312 = AUS ;%{SE}%MKUKATPVW %CVW_SPS %VBOASG %P 2:F312 = AUS, 3: BOASG
         $FLAG[312] = FALSE
      ;ENDFOLD
      ;FOLD F313 = AUS ;%{SE}%MKUKATPVW %CVW_SPS %VBOASG %P 2:F313 = AUS, 3: BOASG
         $FLAG[313] = FALSE
      ;ENDFOLD
      ;FOLD F324 = AUS ;%{SE}%MKUKATPVW %CVW_SPS %VBOASG %P 2:F324 = AUS, 3: BOASG
         $FLAG[324] = FALSE
      ;ENDFOLD
      ;FOLD F328 = AUS ;%{SE}%MKUKATPVW %CVW_SPS %VBOASG %P 2:F328 = AUS, 3: BOASG
         $FLAG[328] = FALSE
      ;ENDFOLD
      ;FOLD -- ServoGun Dress in Positon AUS -- ;%{SE}%MKUKATPVW %CVW_COM %VCOMMENT %P 2:-- ServoGun Dress in Positon AUS --, 3: VW_COMMENT
      ;ENDFOLD
      ;FOLD A3903 = AUS ;%{SE}%MKUKATPVW %CVW_SPS %VBOASG %P 2:A3903 = AUS, 3: BOASG
         $OUT[3903] = FALSE
      ;ENDFOLD
      ;FOLD -- KF1 einschalten nach Fehler -- ;%{SE}%MKUKATPVW %CVW_COM %VCOMMENT %P 2:-- KF1 einschalten nach Fehler --, 3: VW_COMMENT
      ;ENDFOLD
      ;FOLD A994 = EIN ;%{SE}%MKUKATPVW %CVW_SPS %VBOASG %P 2:A994 = EIN, 3: BOASG
         $OUT[994] = TRUE
      ;ENDFOLD
      ;FOLD -- KF1 Versetzeinheit rueck -- ;%{SE}%MKUKATPVW %CVW_COM %VCOMMENT %P 2:-- KF1 Versetzeinheit rueck --, 3: VW_COMMENT
      ;ENDFOLD
      ;FOLD A995 = AUS ;%{SE}%MKUKATPVW %CVW_SPS %VBOASG %P 2:A995 = AUS, 3: BOASG
         $OUT[995] = FALSE
      ;ENDFOLD
      ;FOLD bin30 ( EIN ) = p112 ;%{SE}%MKUKATPVW %CVW_SPS %VARIASG %P 2:bin30 ( EIN ) = p112, 3: ARIASG
         VW(#BINOUT,TRUE,30,PROCPAR[112])
      ;ENDFOLD
      ;FOLD -- Warte bis Fraeser in Position -- ;%{SE}%MKUKATPVW %CVW_COM %VCOMMENT %P 2:-- Warte bis Fraeser in Position --, 3: VW_COMMENT
      ;ENDFOLD
      ;FOLD SCHRITT 213 = !E995 & !E996 & E997 & E998 & !E999 & A4039 ;%{SE}%MKUKATPVW %CVW_SPS %VST_CON %P 2:SCHRITT 213 = !E995 & !E996 & E997 & E998 & !E999 & A4039, 3: ST_CON
         IF NOT $IN[995] AND NOT $IN[996] AND $IN[997] AND $IN[998] AND NOT $IN[999] AND $OUT[4039] THEN
            PREV_STEP[9] = APP_INT_STEP[9]
            APP_INT_STEP[9] = 213
         ENDIF
      ;ENDFOLD
      ;FOLD SCHRITT 213 = T11 & !E996 & E997 & E998 & !E999 & A4039 ;%{SE}%MKUKATPVW %CVW_SPS %VST_CON %P 2:SCHRITT 213 = T11 & !E996 & E997 & E998 & !E999 & A4039, 3: ST_CON
         IF $TIMER_FLAG[11] AND NOT $IN[996] AND $IN[997] AND $IN[998] AND NOT $IN[999] AND $OUT[4039] THEN
            PREV_STEP[9] = APP_INT_STEP[9]
            APP_INT_STEP[9] = 213
         ENDIF
      ;ENDFOLD
   ;ENDFOLD
   ;FOLD SCHRITT 213 -- st. RZ2 # DressInPos -- ;%{P}%MKUKATPVW,%CSTEP,%VST_NR,%P 1:SCHRITT, 2:213, 3: st. RZ2 # DressInPos
      ;FOLD ;%{H}
         Case 213
      ;ENDFOLD
      ;FOLD A1000 = AUS ;%{SE}%MKUKATPVW %CVW_SPS %VBOASG %P 2:A1000 = AUS, 3: BOASG
         $OUT[1000] = FALSE
      ;ENDFOLD
      ;FOLD -- Ueberwachungszeit ServoGun SZ2 schliessen -- ;%{SE}%MKUKATPVW %CVW_COM %VCOMMENT %P 2:-- Ueberwachungszeit ServoGun SZ2 schliessen --, 3: VW_COMMENT
      ;ENDFOLD
      ;FOLD t9 ( EIN ) = -80[1/10Sek] ;%{SE}%MKUKATPVW %CVW_SPS %VTASG %P 2:t9 ( EIN ) = -80[1/10Sek], 3: TASG
         VW(#SET_TIME,TRUE,9,0,-80)
      ;ENDFOLD
      ;FOLD -- Verweilzeit Versetzeinheit Rueck -- ;%{SE}%MKUKATPVW %CVW_COM %VCOMMENT %P 2:-- Verweilzeit Versetzeinheit Rueck --, 3: VW_COMMENT
      ;ENDFOLD
      ;FOLD t11 ( EIN ) = STOP ;%{SE}%MKUKATPVW %CVW_SPS %VTSTOP %P 2:t11 ( EIN ) = STOP, 3: TSTOP
         VW(#SET_TIME,TRUE,11,1,0)
      ;ENDFOLD
      ;FOLD -- ServoGun SZ1 schliessen -- ;%{SE}%MKUKATPVW %CVW_COM %VCOMMENT %P 2:-- ServoGun SZ1 schliessen --, 3: VW_COMMENT
      ;ENDFOLD
      ;FOLD A3903 = !E996 & E997 & E998 & !E999 ;%{SE}%MKUKATPVW %CVW_SPS %VBOASG %P 2:A3903 = !E996 & E997 & E998 & !E999, 3: BOASG
         $OUT[3903] = NOT $IN[996] AND $IN[997] AND $IN[998] AND NOT $IN[999]
      ;ENDFOLD
      ;FOLD -- KF1 Ausblasen -- ;%{SE}%MKUKATPVW %CVW_COM %VCOMMENT %P 2:-- KF1 Ausblasen --, 3: VW_COMMENT
      ;ENDFOLD
      ;FOLD A996 = F330 + F331 + !F330 & !F331 & !F332 ;%{SE}%MKUKATPVW %CVW_SPS %VBOASG %P 2:A996 = F330 + F331 + !F330 & !F331 & !F332, 3: BOASG
         $OUT[996] = $FLAG[330] OR $FLAG[331] OR NOT $FLAG[330] AND NOT $FLAG[331] AND NOT $FLAG[332]
      ;ENDFOLD
      ;FOLD Schritt 214 = !A3894 & A3896 & A4039 + T9 ;%{SE}%MKUKATPVW %CVW_SPS %VST_CON %P 2:Schritt 214 = !A3894 & A3896 & A4039 + T9, 3: ST_CON
         IF NOT $OUT[3894] AND $OUT[3896] AND $OUT[4039] OR $TIMER_FLAG[9] THEN
            PREV_STEP[9] = APP_INT_STEP[9]
            APP_INT_STEP[9] = 214
         ENDIF
      ;ENDFOLD
      ;FOLD Schritt 50 = A3894 & !A3896 & A4039 & A3509 ;%{SE}%MKUKATPVW %CVW_SPS %VST_CON %P 2:Schritt 50 = A3894 & !A3896 & A4039 & A3509, 3: ST_CON
         IF $OUT[3894] AND NOT $OUT[3896] AND $OUT[4039] AND $OUT[3509] THEN
            PREV_STEP[9] = APP_INT_STEP[9]
            APP_INT_STEP[9] = 50
         ENDIF
      ;ENDFOLD
   ;ENDFOLD
   ;FOLD SCHRITT 214 -- st. RZ2 -- ;%{P}%MKUKATPVW,%CSTEP,%VST_NR,%P 1:SCHRITT, 2:214, 3: st. RZ2
      ;FOLD ;%{H}
         Case 214
      ;ENDFOLD
      ;FOLD -- RSK Fehlerausgabe Kraftaufbau -- ;%{SE}%MKUKATPVW %CVW_COM %VCOMMENT %P 2:-- RSK Fehlerausgabe Kraftaufbau --, 3: VW_COMMENT
      ;ENDFOLD
      ;FOLD F325 = T9 ;%{SE}%MKUKATPVW %CVW_SPS %VBOASG %P 2:F325 = T9, 3: BOASG
         $FLAG[325] = $TIMER_FLAG[9]
      ;ENDFOLD
      ;FOLD -- RSK Sammelstoerung -- ;%{SE}%MKUKATPVW %CVW_COM %VCOMMENT %P 2:-- RSK Sammelstoerung --, 3: VW_COMMENT
      ;ENDFOLD
      ;FOLD F329 = F325 ;%{SE}%MKUKATPVW %CVW_SPS %VBOASG %P 2:F329 = F325, 3: BOASG
         $FLAG[329] = $FLAG[325]
      ;ENDFOLD
      ;FOLD -- KF1 abschalten bei Fehler -- ;%{SE}%MKUKATPVW %CVW_COM %VCOMMENT %P 2:-- KF1 abschalten bei Fehler --, 3: VW_COMMENT
      ;ENDFOLD
      ;FOLD A994 = !T9 ;%{SE}%MKUKATPVW %CVW_SPS %VBOASG %P 2:A994 = !T9, 3: BOASG
         $OUT[994] = NOT $TIMER_FLAG[9]
      ;ENDFOLD
      ;FOLD -- KF1 Ausblasen -- ;%{SE}%MKUKATPVW %CVW_COM %VCOMMENT %P 2:-- KF1 Ausblasen --, 3: VW_COMMENT
      ;ENDFOLD
      ;FOLD A996 = (F330 + F331 + !F330 & !F331 & !F332) & !T9 ;%{SE}%MKUKATPVW %CVW_SPS %VBOASG %P 2:A996 = (F330 + F331 + !F330 & !F331 & !F332) & !T9, 3: BOASG
         $OUT[996] = ($FLAG[330] OR $FLAG[331] OR NOT $FLAG[330] AND NOT $FLAG[331] AND NOT $FLAG[332]) AND NOT $TIMER_FLAG[9]
      ;ENDFOLD
      ;FOLD -- Ueberwachungszeit Fehler Fraesen -- ;%{SE}%MKUKATPVW %CVW_COM %VCOMMENT %P 2:-- Ueberwachungszeit Fehler Fraesen --, 3: VW_COMMENT
      ;ENDFOLD
      ;FOLD t11 ( EIN ) = -110 [1/10Sek] ;%{SE}%MKUKATPVW %CVW_SPS %VTASG %P 2:t11 ( EIN ) = -110 [1/10Sek], 3: TASG
         VW(#SET_TIME,TRUE,11,0,-110)
      ;ENDFOLD
      ;FOLD -- Warte Fraesen fertig oder Timeout -- ;%{SE}%MKUKATPVW %CVW_COM %VCOMMENT %P 2:-- Warte Fraesen fertig oder Timeout --, 3: VW_COMMENT
      ;ENDFOLD
      ;FOLD SCHRITT 215 = (F139 & F154 + F138 & F150 & !F287 + T7 + T9 + F325) & A4039 ;%{SE}%MKUKATPVW %CVW_SPS %VST_CON %P 2:SCHRITT 215 = (F139 & F154 + F138 & F150 & !F287 + T7 + T9 + F325) & A4039, 3: ST_CON
         IF ($FLAG[139] AND $FLAG[154] OR $FLAG[138] AND $FLAG[150] AND NOT $FLAG[287] OR $TIMER_FLAG[7] OR $TIMER_FLAG[9] OR $FLAG[325]) AND $OUT[4039] THEN
            PREV_STEP[9] = APP_INT_STEP[9]
            APP_INT_STEP[9] = 215
         ENDIF
      ;ENDFOLD
      ;FOLD SCHRITT 215 = (F138 & F152 & F287 + T7 + T9 + F325) & A4039 ;%{SE}%MKUKATPVW %CVW_SPS %VST_CON %P 2:SCHRITT 215 = (F138 & F152 & F287 + T7 + T9 + F325) & A4039, 3: ST_CON
         IF ($FLAG[138] AND $FLAG[152] AND $FLAG[287] OR $TIMER_FLAG[7] OR $TIMER_FLAG[9] OR $FLAG[325]) AND $OUT[4039] THEN
            PREV_STEP[9] = APP_INT_STEP[9]
            APP_INT_STEP[9] = 215
         ENDIF
      ;ENDFOLD
   ;ENDFOLD
   ;FOLD SCHRITT 215 -- st. RZ2 # GunOpen -- ;%{P}%MKUKATPVW,%CSTEP,%VST_NR,%P 1:SCHRITT, 2:215, 3: st. RZ2 # GunOpen
      ;FOLD ;%{H}
         Case 215
      ;ENDFOLD
      ;FOLD -- ServoGun SZ1 oeffnen -- ;%{SE}%MKUKATPVW %CVW_COM %VCOMMENT %P 2:-- ServoGun SZ1 oeffnen --, 3: VW_COMMENT
      ;ENDFOLD
      ;FOLD t9 ( EIN ) = STOP ;%{SE}%MKUKATPVW %CVW_SPS %VTSTOP %P 2:t9 ( EIN ) = STOP, 3: TSTOP
         VW(#SET_TIME,TRUE,9,1,0)
      ;ENDFOLD
      ;FOLD A3903 = AUS ;%{SE}%MKUKATPVW %CVW_SPS %VBOASG %P 2:A3903 = AUS, 3: BOASG
         $OUT[3903] = FALSE
      ;ENDFOLD
      ;FOLD A3904 = EIN ;%{SE}%MKUKATPVW %CVW_SPS %VBOASG %P 2:A3904 = EIN, 3: BOASG
         $OUT[3904] = TRUE
      ;ENDFOLD
      ;FOLD -- KF1 Ausblasen -- ;%{SE}%MKUKATPVW %CVW_COM %VCOMMENT %P 2:-- KF1 Ausblasen --, 3: VW_COMMENT
      ;ENDFOLD
      ;FOLD A996 = (F330 + F331 + F332 + !F330 & !F331 & !F332) & !T9 ;%{SE}%MKUKATPVW %CVW_SPS %VBOASG %P 2:A996 = (F330 + F331 + F332 + !F330 & !F331 & !F332) & !T9, 3: BOASG
         $OUT[996] = ($FLAG[330] OR $FLAG[331] OR $FLAG[332] OR NOT $FLAG[330] AND NOT $FLAG[331] AND NOT $FLAG[332]) AND NOT $TIMER_FLAG[9]
      ;ENDFOLD
      ;FOLD -- KF Ausblasen Ausschaltverzoegerung starten -- ;%{SE}%MKUKATPVW %CVW_COM %VCOMMENT %P 2:-- KF Ausblasen Ausschaltverzoegerung starten --, 3: VW_COMMENT
      ;ENDFOLD
      ;FOLD F738 = AUS ;%{SE}%MKUKATPVW %CVW_SPS %VBOASG %P 2:F738 = AUS, 3: BOASG
         $FLAG[738] = FALSE
      ;ENDFOLD
      ;FOLD -- RSK Sammelstoerung -- ;%{SE}%MKUKATPVW %CVW_COM %VCOMMENT %P 2:-- RSK Sammelstoerung --, 3: VW_COMMENT
      ;ENDFOLD
      ;FOLD F329 = T7 + T9 + F325 ;%{SE}%MKUKATPVW %CVW_SPS %VBOASG %P 2:F329 = T7 + T9 + F325, 3: BOASG
         $FLAG[329] = $TIMER_FLAG[7] OR $TIMER_FLAG[9] OR $FLAG[325]
      ;ENDFOLD
      ;FOLD -- Hilfsflag Startfraesen -- ;%{SE}%MKUKATPVW %CVW_COM %VCOMMENT %P 2:-- Hilfsflag Startfraesen --, 3: VW_COMMENT
      ;ENDFOLD
      ;FOLD F152 = F152 & F287 ;%{SE}%MKUKATPVW %CVW_SPS %VBOASG %P 2:F152 = F152 & F287, 3: BOASG
         $FLAG[152] = $FLAG[152] AND $FLAG[287]
      ;ENDFOLD
      ;FOLD F152 = (F152 & F138 + F154 & F139) & F287 ;%{SE}%MKUKATPVW %CVW_SPS %VBOASG %P 2:F152 = (F152 & F138 + F154 & F139) & F287, 3: BOASG
         $FLAG[152] = ($FLAG[152] AND $FLAG[138] OR $FLAG[154] AND $FLAG[139]) AND $FLAG[287]
      ;ENDFOLD
      ;FOLD F154 = !F130 & F154 + F130 & F287 & F154 ;%{SE}%MKUKATPVW %CVW_SPS %VBOASG %P 2:F154 = !F130 & F154 + F130 & F287 & F154, 3: BOASG
         $FLAG[154] = NOT $FLAG[130] AND $FLAG[154] OR $FLAG[130] AND $FLAG[287] AND $FLAG[154]
      ;ENDFOLD
      ;FOLD F287 = F138 + F139 & F130 ;%{SE}%MKUKATPVW %CVW_SPS %VBOASG %P 2:F287 = F138 + F139 & F130, 3: BOASG
         $FLAG[287] = $FLAG[138] OR $FLAG[139] AND $FLAG[130]
      ;ENDFOLD
      ;FOLD -- Neues Fraesprogramm und Zaehler ruecksetzen -- ;%{SE}%MKUKATPVW %CVW_COM %VCOMMENT %P 2:-- Neues Fraesprogramm und Zaehler ruecksetzen --, 3: VW_COMMENT
      ;ENDFOLD
      ;FOLD bin31 ( F164 ) = 36 ;%{SE}%MKUKATPVW %CVW_SPS %VARIASG %P 2:bin31 ( F164 ) = 36, 3: ARIASG
         VW(#BINOUT,$FLAG[164],31,36)
      ;ENDFOLD
      ;FOLD i7 ( F152 ) = i45 ;%{SE}%MKUKATPVW %CVW_SPS %VARIASG %P 2:i7 ( F152 ) = i45, 3: ARIASG
         VW(#COUNTER,$FLAG[152],7,$COUNT_I[45])
      ;ENDFOLD
      ;FOLD -- Fehler Fraesen -- ;%{SE}%MKUKATPVW %CVW_COM %VCOMMENT %P 2:-- Fehler Fraesen --, 3: VW_COMMENT
      ;ENDFOLD
      ;FOLD Schritt 250 = (!A3894 & !A3508 & T11) + (A3894 & !A3508 & T11) & A4039 ;%{SE}%MKUKATPVW %CVW_SPS %VST_CON %P 2:Schritt 250 = (!A3894 & !A3508 & T11) + (A3894 & !A3508 & T11) & A4039, 3: ST_CON
         IF (NOT $OUT[3894] AND NOT $OUT[3508] AND $TIMER_FLAG[11]) OR ($OUT[3894] AND NOT $OUT[3508] AND $TIMER_FLAG[11]) AND $OUT[4039] THEN
            PREV_STEP[9] = APP_INT_STEP[9]
            APP_INT_STEP[9] = 250
         ENDIF
      ;ENDFOLD
      ;FOLD -- Wiederholung beim Normalfraesen -- ;%{SE}%MKUKATPVW %CVW_COM %VCOMMENT %P 2:-- Wiederholung beim Normalfraesen --, 3: VW_COMMENT
      ;ENDFOLD
      ;FOLD Schritt 211 = A3894 & A3508 & (!F138 & F139 & F130 & !F152) & !F329 & A4039 ;%{SE}%MKUKATPVW %CVW_SPS %VST_CON %P 2:Schritt 211 = A3894 & A3508 & (!F138 & F139 & F130 & !F152) & !F329 & A4039, 3: ST_CON
         IF $OUT[3894] AND $OUT[3508] AND (NOT $FLAG[138] AND $FLAG[139] AND $FLAG[130] AND NOT $FLAG[152]) AND NOT $FLAG[329] AND $OUT[4039] THEN
            PREV_STEP[9] = APP_INT_STEP[9]
            APP_INT_STEP[9] = 211
         ENDIF
      ;ENDFOLD
      ;FOLD -- Wiederholung beim Startfraesen -- ;%{SE}%MKUKATPVW %CVW_COM %VCOMMENT %P 2:-- Wiederholung beim Startfraesen --, 3: VW_COMMENT
      ;ENDFOLD
      ;FOLD Schritt 211 = A3894 & A3508 & (F138 & !F152 + F139 & F130 & !F152) & !F329 & A4039 & A3520 ;%{SE}%MKUKATPVW %CVW_SPS %VST_CON %P 2:Schritt 211 = A3894 & A3508 & (F138 & !F152 + F139 & F130 & !F152) & !F329 & A4039 & A3520, 3: ST_CON
         IF $OUT[3894] AND $OUT[3508] AND ($FLAG[138] AND NOT $FLAG[152] OR $FLAG[139] AND $FLAG[130] AND NOT $FLAG[152]) AND NOT $FLAG[329] AND $OUT[4039] AND $OUT[3520] THEN
            PREV_STEP[9] = APP_INT_STEP[9]
            APP_INT_STEP[9] = 211
         ENDIF
      ;ENDFOLD
      ;FOLD -- Wiederholung beim Startfraesen -- ;%{SE}%MKUKATPVW %CVW_COM %VCOMMENT %P 2:-- Wiederholung beim Startfraesen --, 3: VW_COMMENT
      ;ENDFOLD
      ;FOLD Schritt 216 = A3894 & A3508 & (F138 & !F152 + F139 & F130 & F152) & !F329 & A4039 & !A3520 ;%{SE}%MKUKATPVW %CVW_SPS %VST_CON %P 2:Schritt 216 = A3894 & A3508 & (F138 & !F152 + F139 & F130 & F152) & !F329 & A4039 & !A3520, 3: ST_CON
         IF $OUT[3894] AND $OUT[3508] AND ($FLAG[138] AND NOT $FLAG[152] OR $FLAG[139] AND $FLAG[130] AND $FLAG[152]) AND NOT $FLAG[329] AND $OUT[4039] AND NOT $OUT[3520] THEN
            PREV_STEP[9] = APP_INT_STEP[9]
            APP_INT_STEP[9] = 216
         ENDIF
      ;ENDFOLD
      ;FOLD -- Weiter wenn Fraesen fertig -- ;%{SE}%MKUKATPVW %CVW_COM %VCOMMENT %P 2:-- Weiter wenn Fraesen fertig --, 3: VW_COMMENT
      ;ENDFOLD
      ;FOLD Schritt 216 = A3894 & A3508 & (F139 & F154 & (!F130 + F152) + F138 & F152 + F329) & A4039 ;%{SE}%MKUKATPVW %CVW_SPS %VST_CON %P 2:Schritt 216 = A3894 & A3508 & (F139 & F154 & (!F130 + F152) + F138 & F152 + F329) & A4039, 3: ST_CON
         IF $OUT[3894] AND $OUT[3508] AND ($FLAG[139] AND $FLAG[154] AND (NOT $FLAG[130] OR $FLAG[152]) OR $FLAG[138] AND $FLAG[152] OR $FLAG[329]) AND $OUT[4039] THEN
            PREV_STEP[9] = APP_INT_STEP[9]
            APP_INT_STEP[9] = 216
         ENDIF
      ;ENDFOLD
   ;ENDFOLD
   ;FOLD SCHRITT 216 -- st. RZ2 # StartAcknowledge -- ;%{P}%MKUKATPVW,%CSTEP,%VST_NR,%P 1:SCHRITT, 2:216, 3: st. RZ2 # StartAcknowledge
      ;FOLD ;%{H}
         Case 216
      ;ENDFOLD
      ;FOLD -- Hilfsflag Durchlaufmerker -- ;%{SE}%MKUKATPVW %CVW_COM %VCOMMENT %P 2:-- Hilfsflag Durchlaufmerker --, 3: VW_COMMENT
      ;ENDFOLD
      ;FOLD F324 = AUS ;%{SE}%MKUKATPVW %CVW_SPS %VBOASG %P 2:F324 = AUS, 3: BOASG
         $FLAG[324] = FALSE
      ;ENDFOLD
      ;FOLD A3903 = AUS ;%{SE}%MKUKATPVW %CVW_SPS %VBOASG %P 2:A3903 = AUS, 3: BOASG
         $OUT[3903] = FALSE
      ;ENDFOLD
      ;FOLD A3904 = AUS ;%{SE}%MKUKATPVW %CVW_SPS %VBOASG %P 2:A3904 = AUS, 3: BOASG
         $OUT[3904] = FALSE
      ;ENDFOLD
      ;FOLD A3510 = AUS ;%{SE}%MKUKATPVW %CVW_SPS %VBOASG %P 2:A3510 = AUS, 3: BOASG
         $OUT[3510] = FALSE
      ;ENDFOLD
      ;FOLD A3512 = EIN ;%{SE}%MKUKATPVW %CVW_SPS %VBOASG %P 2:A3512 = EIN, 3: BOASG
         $OUT[3512] = TRUE
      ;ENDFOLD
      ;FOLD t9 ( EIN ) = STOP ;%{SE}%MKUKATPVW %CVW_SPS %VTSTOP %P 2:t9 ( EIN ) = STOP, 3: TSTOP
         VW(#SET_TIME,TRUE,9,1,0)
      ;ENDFOLD
      ;FOLD -- KF1 abschalten -- ;%{SE}%MKUKATPVW %CVW_COM %VCOMMENT %P 2:-- KF1 abschalten --, 3: VW_COMMENT
      ;ENDFOLD
      ;FOLD A994 = AUS ;%{SE}%MKUKATPVW %CVW_SPS %VBOASG %P 2:A994 = AUS, 3: BOASG
         $OUT[994] = FALSE
      ;ENDFOLD
      ;FOLD -- Ueberwachungszeit KF1 Versetzeinheit -- ;%{SE}%MKUKATPVW %CVW_COM %VCOMMENT %P 2:-- Ueberwachungszeit KF1 Versetzeinheit --, 3: VW_COMMENT
      ;ENDFOLD
      ;FOLD t8 ( EIN ) = -40[1/10Sek] ;%{SE}%MKUKATPVW %CVW_SPS %VTASG %P 2:t8 ( EIN ) = -40[1/10Sek], 3: TASG
         VW(#SET_TIME,TRUE,8,0,-40)
      ;ENDFOLD
      ;FOLD SCHRITT 217 = A4039 & !E195 ;%{SE}%MKUKATPVW %CVW_SPS %VST_CON %P 2:SCHRITT 217 = A4039 & !E195, 3: ST_CON
         IF $OUT[4039] AND NOT $IN[195] THEN
            PREV_STEP[9] = APP_INT_STEP[9]
            APP_INT_STEP[9] = 217
         ENDIF
      ;ENDFOLD
   ;ENDFOLD
   ;FOLD SCHRITT 217 -- st. RZ2 -- ;%{P}%MKUKATPVW,%CSTEP,%VST_NR,%P 1:SCHRITT, 2:217, 3: st. RZ2
      ;FOLD ;%{H}
         Case 217
      ;ENDFOLD
      ;FOLD -- RSK Fehlerausgabe Arbeitsst. -- ;%{SE}%MKUKATPVW %CVW_COM %VCOMMENT %P 2:-- RSK Fehlerausgabe Arbeitsst. --, 3: VW_COMMENT
      ;ENDFOLD
      ;FOLD F328 = AUS ;%{SE}%MKUKATPVW %CVW_SPS %VBOASG %P 2:F328 = AUS, 3: BOASG
         $FLAG[328] = FALSE
      ;ENDFOLD
      ;FOLD -- KF1 Versetzeinheit vor -- ;%{SE}%MKUKATPVW %CVW_COM %VCOMMENT %P 2:-- KF1 Versetzeinheit vor --, 3: VW_COMMENT
      ;ENDFOLD
      ;FOLD A995 = F564 ;%{SE}%MKUKATPVW %CVW_SPS %VBOASG %P 2:A995 = F564, 3: BOASG
         $OUT[995] = $FLAG[564]
      ;ENDFOLD
      ;FOLD A3512 = AUS ;%{SE}%MKUKATPVW %CVW_SPS %VBOASG %P 2:A3512 = AUS, 3: BOASG
         $OUT[3512] = FALSE
      ;ENDFOLD
      ;FOLD -- RSK Fehlerausgabe KS1 Arbeitsst. -- ;%{SE}%MKUKATPVW %CVW_COM %VCOMMENT %P 2:-- RSK Fehlerausgabe KS1 Arbeitsst. --, 3: VW_COMMENT
      ;ENDFOLD
      ;FOLD F324 = (E996 + !E997 + !E998 + E999) & !F323 & !F328 + F324 ;%{SE}%MKUKATPVW %CVW_SPS %VBOASG %P 2:F324 = (E996 + !E997 + !E998 + E999) & !F323 & !F328 + F324, 3: BOASG
         $FLAG[324] = ($IN[996] OR NOT $IN[997] OR NOT $IN[998] OR $IN[999]) AND NOT $FLAG[323] AND NOT $FLAG[328] OR $FLAG[324]
      ;ENDFOLD
      ;FOLD -- RSK Sammelstoerung -- ;%{SE}%MKUKATPVW %CVW_COM %VCOMMENT %P 2:-- RSK Sammelstoerung --, 3: VW_COMMENT
      ;ENDFOLD
      ;FOLD F329 = F324 + F325 ;%{SE}%MKUKATPVW %CVW_SPS %VBOASG %P 2:F329 = F324 + F325, 3: BOASG
         $FLAG[329] = $FLAG[324] OR $FLAG[325]
      ;ENDFOLD
      ;FOLD -- Ueberwachungszeit KS1 schwenken -- ;%{SE}%MKUKATPVW %CVW_COM %VCOMMENT %P 2:-- Ueberwachungszeit KS1 schwenken --, 3: VW_COMMENT
      ;ENDFOLD
      ;FOLD t9 ( EIN ) = -100[1/10Sek] ;%{SE}%MKUKATPVW %CVW_SPS %VTASG %P 2:t9 ( EIN ) = -100[1/10Sek], 3: TASG
         VW(#SET_TIME,TRUE,9,0,-100)
      ;ENDFOLD
      ;FOLD SCHRITT 216 = F324 & (E26 + E27) & A4039 ;%{SE}%MKUKATPVW %CVW_SPS %VST_CON %P 2:SCHRITT 216 = F324 & (E26 + E27) & A4039, 3: ST_CON
         IF $FLAG[324] AND ($IN[26] OR $IN[27]) AND $OUT[4039] THEN
            PREV_STEP[9] = APP_INT_STEP[9]
            APP_INT_STEP[9] = 216
         ENDIF
      ;ENDFOLD
      ;FOLD SCHRITT 218 = (!F324 & (E995 & F564 + !E995 & !F564) + T8 + F325) & A4039 ;%{SE}%MKUKATPVW %CVW_SPS %VST_CON %P 2:SCHRITT 218 = (!F324 & (E995 & F564 + !E995 & !F564) + T8 + F325) & A4039, 3: ST_CON
         IF (NOT $FLAG[324] AND ($IN[995] AND $FLAG[564] OR NOT $IN[995] AND NOT $FLAG[564]) OR $TIMER_FLAG[8] OR $FLAG[325]) AND $OUT[4039] THEN
            PREV_STEP[9] = APP_INT_STEP[9]
            APP_INT_STEP[9] = 218
         ENDIF
      ;ENDFOLD
   ;ENDFOLD
   ;FOLD SCHRITT 218 -- st. RZ2 # KS in RS schwenken -- ;%{P}%MKUKATPVW,%CSTEP,%VST_NR,%P 1:SCHRITT, 2:218, 3: st. RZ2 # KS in RS schwenken
      ;FOLD ;%{H}
         Case 218
      ;ENDFOLD
      ;FOLD F323 = AUS ;%{SE}%MKUKATPVW %CVW_SPS %VBOASG %P 2:F323 = AUS, 3: BOASG
         $FLAG[323] = FALSE
      ;ENDFOLD
      ;FOLD F328 = AUS ;%{SE}%MKUKATPVW %CVW_SPS %VBOASG %P 2:F328 = AUS, 3: BOASG
         $FLAG[328] = FALSE
      ;ENDFOLD
      ;FOLD -- RSK Sammelstoerung -- ;%{SE}%MKUKATPVW %CVW_COM %VCOMMENT %P 2:-- RSK Sammelstoerung --, 3: VW_COMMENT
      ;ENDFOLD
      ;FOLD F329 = F325 ;%{SE}%MKUKATPVW %CVW_SPS %VBOASG %P 2:F329 = F325, 3: BOASG
         $FLAG[329] = $FLAG[325]
      ;ENDFOLD
      ;FOLD -- KF1 ein -- ;%{SE}%MKUKATPVW %CVW_COM %VCOMMENT %P 2:-- KF1 ein --, 3: VW_COMMENT
      ;ENDFOLD
      ;FOLD A994 = EIN ;%{SE}%MKUKATPVW %CVW_SPS %VBOASG %P 2:A994 = EIN, 3: BOASG
         $OUT[994] = TRUE
      ;ENDFOLD
      ;FOLD -- KF Ausblasen Ausschaltverzoegerung starten -- ;%{SE}%MKUKATPVW %CVW_COM %VCOMMENT %P 2:-- KF Ausblasen Ausschaltverzoegerung starten --, 3: VW_COMMENT
      ;ENDFOLD
      ;FOLD F738 = EIN ;%{SE}%MKUKATPVW %CVW_SPS %VBOASG %P 2:F738 = EIN, 3: BOASG
         $FLAG[738] = TRUE
      ;ENDFOLD
      ;FOLD -- KF1 Ausblasen -- ;%{SE}%MKUKATPVW %CVW_COM %VCOMMENT %P 2:-- KF1 Ausblasen --, 3: VW_COMMENT
      ;ENDFOLD
      ;FOLD A996 = (F330 + F331 + F332) & F738 ;%{SE}%MKUKATPVW %CVW_SPS %VBOASG %P 2:A996 = (F330 + F331 + F332) & F738, 3: BOASG
         $OUT[996] = ($FLAG[330] OR $FLAG[331] OR $FLAG[332]) AND $FLAG[738]
      ;ENDFOLD
      ;FOLD -- KS1 in Ruhestellung schwenken -- ;%{SE}%MKUKATPVW %CVW_COM %VCOMMENT %P 2:-- KS1 in Ruhestellung schwenken --, 3: VW_COMMENT
      ;ENDFOLD
      ;FOLD A1000 = A3894 & (E995 & F564 + !E995 & !F564) ;%{SE}%MKUKATPVW %CVW_SPS %VBOASG %P 2:A1000 = A3894 & (E995 & F564 + !E995 & !F564), 3: BOASG
         $OUT[1000] = $OUT[3894] AND ($IN[995] AND $FLAG[564] OR NOT $IN[995] AND NOT $FLAG[564])
      ;ENDFOLD
      ;FOLD Schritt 220 = A3894 & A1000 & A4039 + T9 ;%{SE}%MKUKATPVW %CVW_SPS %VST_CON %P 2:Schritt 220 = A3894 & A1000 & A4039 + T9, 3: ST_CON
         IF $OUT[3894] AND $OUT[1000] AND $OUT[4039] OR $TIMER_FLAG[9] THEN
            PREV_STEP[9] = APP_INT_STEP[9]
            APP_INT_STEP[9] = 220
         ENDIF
      ;ENDFOLD
   ;ENDFOLD
   ;FOLD SCHRITT 220 -- st. RZ2 -- ;%{P}%MKUKATPVW,%CSTEP,%VST_NR,%P 1:SCHRITT, 2:220, 3: st. RZ2
      ;FOLD ;%{H}
         Case 220
      ;ENDFOLD
      ;FOLD -- Hilfsflag SK Programmwechsel -- ;%{SE}%MKUKATPVW %CVW_COM %VCOMMENT %P 2:-- Hilfsflag SK Programmwechsel --, 3: VW_COMMENT
      ;ENDFOLD
      ;FOLD F334 = AUS ;%{SE}%MKUKATPVW %CVW_SPS %VBOASG %P 2:F334 = AUS, 3: BOASG
         $FLAG[334] = FALSE
      ;ENDFOLD
      ;FOLD -- RSK Fehlerausgabe KF Versetzeinheit -- ;%{SE}%MKUKATPVW %CVW_COM %VCOMMENT %P 2:-- RSK Fehlerausgabe KF Versetzeinheit --, 3: VW_COMMENT
      ;ENDFOLD
      ;FOLD F328 = !E995 & F564 & !F323 + F328 ;%{SE}%MKUKATPVW %CVW_SPS %VBOASG %P 2:F328 = !E995 & F564 & !F323 + F328, 3: BOASG
         $FLAG[328] = NOT $IN[995] AND $FLAG[564] AND NOT $FLAG[323] OR $FLAG[328]
      ;ENDFOLD
      ;FOLD -- RSK Fehlerausgabe KS1 Ruhestellung -- ;%{SE}%MKUKATPVW %CVW_COM %VCOMMENT %P 2:-- RSK Fehlerausgabe KS1 Ruhestellung --, 3: VW_COMMENT
      ;ENDFOLD
      ;FOLD F323 = (!E996 + E997 + E998 + !E999) & T9 & (E995 + !F564) + F323 ;%{SE}%MKUKATPVW %CVW_SPS %VBOASG %P 2:F323 = (!E996 + E997 + E998 + !E999) & T9 & (E995 + !F564) + F323, 3: BOASG
         $FLAG[323] = (NOT $IN[996] OR $IN[997] OR $IN[998] OR NOT $IN[999]) AND $TIMER_FLAG[9] AND ($IN[995] OR NOT $FLAG[564]) OR $FLAG[323]
      ;ENDFOLD
      ;FOLD -- RSK Fehlerausgabe EZ/SP min. Oeffnung -- ;%{SE}%MKUKATPVW %CVW_COM %VCOMMENT %P 2:-- RSK Fehlerausgabe EZ/SP min. Oeffnung --, 3: VW_COMMENT
      ;ENDFOLD
      ;FOLD F333 = !A3894 ;%{SE}%MKUKATPVW %CVW_SPS %VBOASG %P 2:F333 = !A3894, 3: BOASG
         $FLAG[333] = NOT $OUT[3894]
      ;ENDFOLD
      ;FOLD -- RSK Sammelstoerung -- ;%{SE}%MKUKATPVW %CVW_COM %VCOMMENT %P 2:-- RSK Sammelstoerung --, 3: VW_COMMENT
      ;ENDFOLD
      ;FOLD F329 = F323 + F325 + F328 + F333 ;%{SE}%MKUKATPVW %CVW_SPS %VBOASG %P 2:F329 = F323 + F325 + F328 + F333, 3: BOASG
         $FLAG[329] = $FLAG[323] OR $FLAG[325] OR $FLAG[328] OR $FLAG[333]
      ;ENDFOLD
      ;FOLD A994 = !F329 ;%{SE}%MKUKATPVW %CVW_SPS %VBOASG %P 2:A994 = !F329, 3: BOASG
         $OUT[994] = NOT $FLAG[329]
      ;ENDFOLD
      ;FOLD A995 = F564 ;%{SE}%MKUKATPVW %CVW_SPS %VBOASG %P 2:A995 = F564, 3: BOASG
         $OUT[995] = $FLAG[564]
      ;ENDFOLD
      ;FOLD SCHRITT 216 = (F323 + F328) & (E26 + E27) & A4039 ;%{SE}%MKUKATPVW %CVW_SPS %VST_CON %P 2:SCHRITT 216 = (F323 + F328) & (E26 + E27) & A4039, 3: ST_CON
         IF ($FLAG[323] OR $FLAG[328]) AND ($IN[26] OR $IN[27]) AND $OUT[4039] THEN
            PREV_STEP[9] = APP_INT_STEP[9]
            APP_INT_STEP[9] = 216
         ENDIF
      ;ENDFOLD
      ;FOLD SCHRITT 221 = !A1000 & E996 & !E997 & !E998 & E999 & A4039 ;%{SE}%MKUKATPVW %CVW_SPS %VST_CON %P 2:SCHRITT 221 = !A1000 & E996 & !E997 & !E998 & E999 & A4039, 3: ST_CON
         IF NOT $OUT[1000] AND $IN[996] AND NOT $IN[997] AND NOT $IN[998] AND $IN[999] AND $OUT[4039] THEN
            PREV_STEP[9] = APP_INT_STEP[9]
            APP_INT_STEP[9] = 221
         ENDIF
      ;ENDFOLD
   ;ENDFOLD
   ;FOLD SCHRITT 221 -- st. RZ2 -- ;%{P}%MKUKATPVW,%CSTEP,%VST_NR,%P 1:SCHRITT, 2:221, 3: st. RZ2
      ;FOLD ;%{H}
         Case 221
      ;ENDFOLD
      ;FOLD A1000 = AUS ;%{SE}%MKUKATPVW %CVW_SPS %VBOASG %P 2:A1000 = AUS, 3: BOASG
         $OUT[1000] = FALSE
      ;ENDFOLD
      ;FOLD F323 = AUS ;%{SE}%MKUKATPVW %CVW_SPS %VBOASG %P 2:F323 = AUS, 3: BOASG
         $FLAG[323] = FALSE
      ;ENDFOLD
      ;FOLD F328 = AUS ;%{SE}%MKUKATPVW %CVW_SPS %VBOASG %P 2:F328 = AUS, 3: BOASG
         $FLAG[328] = FALSE
      ;ENDFOLD
      ;FOLD -- KF Ausblasen Ausschaltverzoegerung starten -- ;%{SE}%MKUKATPVW %CVW_COM %VCOMMENT %P 2:-- KF Ausblasen Ausschaltverzoegerung starten --, 3: VW_COMMENT
      ;ENDFOLD
      ;FOLD F738 = EIN ;%{SE}%MKUKATPVW %CVW_SPS %VBOASG %P 2:F738 = EIN, 3: BOASG
         $FLAG[738] = TRUE
      ;ENDFOLD
      ;FOLD -- RSK Sammelstoerung -- ;%{SE}%MKUKATPVW %CVW_COM %VCOMMENT %P 2:-- RSK Sammelstoerung --, 3: VW_COMMENT
      ;ENDFOLD
      ;FOLD F329 = F325 ;%{SE}%MKUKATPVW %CVW_SPS %VBOASG %P 2:F329 = F325, 3: BOASG
         $FLAG[329] = $FLAG[325]
      ;ENDFOLD
      ;FOLD t9 ( EIN ) = STOP ;%{SE}%MKUKATPVW %CVW_SPS %VTSTOP %P 2:t9 ( EIN ) = STOP, 3: TSTOP
         VW(#SET_TIME,TRUE,9,1,0)
      ;ENDFOLD
      ;FOLD -- KF1 Versetzeinheit rueck -- ;%{SE}%MKUKATPVW %CVW_COM %VCOMMENT %P 2:-- KF1 Versetzeinheit rueck --, 3: VW_COMMENT
      ;ENDFOLD
      ;FOLD A995 = AUS ;%{SE}%MKUKATPVW %CVW_SPS %VBOASG %P 2:A995 = AUS, 3: BOASG
         $OUT[995] = FALSE
      ;ENDFOLD
      ;FOLD -- KF1 aus -- ;%{SE}%MKUKATPVW %CVW_COM %VCOMMENT %P 2:-- KF1 aus --, 3: VW_COMMENT
      ;ENDFOLD
      ;FOLD A994 = AUS ;%{SE}%MKUKATPVW %CVW_SPS %VBOASG %P 2:A994 = AUS, 3: BOASG
         $OUT[994] = FALSE
      ;ENDFOLD
      ;FOLD -- KF1 Ausblasen -- ;%{SE}%MKUKATPVW %CVW_COM %VCOMMENT %P 2:-- KF1 Ausblasen --, 3: VW_COMMENT
      ;ENDFOLD
      ;FOLD A996 = (F330 + F331 + F332) & F738 ;%{SE}%MKUKATPVW %CVW_SPS %VBOASG %P 2:A996 = (F330 + F331 + F332) & F738, 3: BOASG
         $OUT[996] = ($FLAG[330] OR $FLAG[331] OR $FLAG[332]) AND $FLAG[738]
      ;ENDFOLD
      ;FOLD bin4 ( !F329 ) = 1 ;%{SE}%MKUKATPVW %CVW_SPS %VARIASG %P 2:bin4 ( !F329 ) = 1, 3: ARIASG
         VW(#BINOUT,NOT $FLAG[329],4,1)
      ;ENDFOLD
      ;FOLD bin6 ( !F329 ) = 1 ;%{SE}%MKUKATPVW %CVW_SPS %VARIASG %P 2:bin6 ( !F329 ) = 1, 3: ARIASG
         VW(#BINOUT,NOT $FLAG[329],6,1)
      ;ENDFOLD
      ;FOLD bin31 ( !F329 ) = 1 ;%{SE}%MKUKATPVW %CVW_SPS %VARIASG %P 2:bin31 ( !F329 ) = 1, 3: ARIASG
         VW(#BINOUT,NOT $FLAG[329],31,1)
      ;ENDFOLD
      ;FOLD -- Wartezeit Programmwechsel SK -- ;%{SE}%MKUKATPVW %CVW_COM %VCOMMENT %P 2:-- Wartezeit Programmwechsel SK --, 3: VW_COMMENT
      ;ENDFOLD
      ;FOLD T8 ( !F334 ) = -2[1/10Sek] ;%{SE}%MKUKATPVW %CVW_SPS %VTASG %P 2:T8 ( !F334 ) = -2[1/10Sek], 3: TASG
         VW(#SET_TIME,NOT $FLAG[334],8,0,-2)
      ;ENDFOLD
      ;FOLD -- Hilfsflag SK Programmwechsel -- ;%{SE}%MKUKATPVW %CVW_COM %VCOMMENT %P 2:-- Hilfsflag SK Programmwechsel --, 3: VW_COMMENT
      ;ENDFOLD
      ;FOLD F334 = EIN ;%{SE}%MKUKATPVW %CVW_SPS %VBOASG %P 2:F334 = EIN, 3: BOASG
         $FLAG[334] = TRUE
      ;ENDFOLD
      ;FOLD SCHRITT 203 = (F325 + F329) & (E26 + E27) & A4039 ;%{SE}%MKUKATPVW %CVW_SPS %VST_CON %P 2:SCHRITT 203 = (F325 + F329) & (E26 + E27) & A4039, 3: ST_CON
         IF ($FLAG[325] OR $FLAG[329]) AND ($IN[26] OR $IN[27]) AND $OUT[4039] THEN
            PREV_STEP[9] = APP_INT_STEP[9]
            APP_INT_STEP[9] = 203
         ENDIF
      ;ENDFOLD
      ;FOLD SCHRITT 222 = T8 & !F325 & !F329 & A4039 & (A3506 & A3505) ;%{SE}%MKUKATPVW %CVW_SPS %VST_CON %P 2:SCHRITT 222 = T8 & !F325 & !F329 & A4039 & (A3506 & A3505), 3: ST_CON
         IF $TIMER_FLAG[8] AND NOT $FLAG[325] AND NOT $FLAG[329] AND $OUT[4039] AND ($OUT[3506] AND $OUT[3505]) THEN
            PREV_STEP[9] = APP_INT_STEP[9]
            APP_INT_STEP[9] = 222
         ENDIF
      ;ENDFOLD
   ;ENDFOLD
   ;FOLD SCHRITT 222 -- st. RZ2 -- ;%{P}%MKUKATPVW,%CSTEP,%VST_NR,%P 1:SCHRITT, 2:222, 3: st. RZ2
      ;FOLD ;%{H}
         Case 222
      ;ENDFOLD
      ;FOLD -- Hilfsflag SK Programmwechsel -- ;%{SE}%MKUKATPVW %CVW_COM %VCOMMENT %P 2:-- Hilfsflag SK Programmwechsel --, 3: VW_COMMENT
      ;ENDFOLD
      ;FOLD F334 = AUS ;%{SE}%MKUKATPVW %CVW_SPS %VBOASG %P 2:F334 = AUS, 3: BOASG
         $FLAG[334] = FALSE
      ;ENDFOLD
      ;FOLD -- Quitt. Fraesen SK1 -- ;%{SE}%MKUKATPVW %CVW_COM %VCOMMENT %P 2:-- Quitt. Fraesen SK1 --, 3: VW_COMMENT
      ;ENDFOLD
      ;FOLD A946 = (!F322 & !F830) + (F830 & A946) + (E193 + A3505) & EIN ;%{SE}%MKUKATPVW %CVW_SPS %VBOASG %P 2:A946 = (!F322 & !F830) + (F830 & A946) + (E193 + A3505) & EIN, 3: BOASG
         $OUT[946] = (NOT $FLAG[322] AND NOT $FLAG[830]) OR ($FLAG[830] AND $OUT[946]) OR ($IN[193] OR $OUT[3505]) AND TRUE
      ;ENDFOLD
      ;FOLD A3904 = (!F138 & F139 & !F830) + (F830 & A3904) ;%{SE}%MKUKATPVW %CVW_SPS %VBOASG %P 2:A3904 = (!F138 & F139 & !F830) + (F830 & A3904), 3: BOASG
         $OUT[3904] = (NOT $FLAG[138] AND $FLAG[139] AND NOT $FLAG[830]) OR ($FLAG[830] AND $OUT[3904])
      ;ENDFOLD
      ;FOLD A3512 = (F138 & !F139 & !F830) + (F830 & A3512) ;%{SE}%MKUKATPVW %CVW_SPS %VBOASG %P 2:A3512 = (F138 & !F139 & !F830) + (F830 & A3512), 3: BOASG
         $OUT[3512] = ($FLAG[138] AND NOT $FLAG[139] AND NOT $FLAG[830]) OR ($FLAG[830] AND $OUT[3512])
      ;ENDFOLD
      ;FOLD SCHRITT 223 = A4039 & (!E946 & !E948 & !F830) ;%{SE}%MKUKATPVW %CVW_SPS %VST_CON %P 2:SCHRITT 223 = A4039 & (!E946 & !E948 & !F830), 3: ST_CON
         IF $OUT[4039] AND (NOT $IN[946] AND NOT $IN[948] AND NOT $FLAG[830]) THEN
            PREV_STEP[9] = APP_INT_STEP[9]
            APP_INT_STEP[9] = 223
         ENDIF
      ;ENDFOLD
   ;ENDFOLD
   ;FOLD SCHRITT 223 -- st. RZ2 # Ruecksetzen -- ;%{P}%MKUKATPVW,%CSTEP,%VST_NR,%P 1:SCHRITT, 2:223, 3: st. RZ2 # Ruecksetzen
      ;FOLD ;%{H}
         Case 223
      ;ENDFOLD
      ;FOLD -- Start Init Same AUS -- ;%{SE}%MKUKATPVW %CVW_COM %VCOMMENT %P 2:-- Start Init Same AUS --, 3: VW_COMMENT
      ;ENDFOLD
      ;FOLD A3514 = AUS ;%{SE}%MKUKATPVW %CVW_SPS %VBOASG %P 2:A3514 = AUS, 3: BOASG
         $OUT[3514] = FALSE
      ;ENDFOLD
      ;FOLD -- Start Spot AUS -- ;%{SE}%MKUKATPVW %CVW_COM %VCOMMENT %P 2:-- Start Spot AUS --, 3: VW_COMMENT
      ;ENDFOLD
      ;FOLD A3511 = AUS ;%{SE}%MKUKATPVW %CVW_SPS %VBOASG %P 2:A3511 = AUS, 3: BOASG
         $OUT[3511] = FALSE
      ;ENDFOLD
      ;FOLD -- Start Dress AUS -- ;%{SE}%MKUKATPVW %CVW_COM %VCOMMENT %P 2:-- Start Dress AUS --, 3: VW_COMMENT
      ;ENDFOLD
      ;FOLD A3510 = AUS ;%{SE}%MKUKATPVW %CVW_SPS %VBOASG %P 2:A3510 = AUS, 3: BOASG
         $OUT[3510] = FALSE
      ;ENDFOLD
      ;FOLD -- Start Init New AUS -- ;%{SE}%MKUKATPVW %CVW_COM %VCOMMENT %P 2:-- Start Init New AUS --, 3: VW_COMMENT
      ;ENDFOLD
      ;FOLD A3513 = AUS ;%{SE}%MKUKATPVW %CVW_SPS %VBOASG %P 2:A3513 = AUS, 3: BOASG
         $OUT[3513] = FALSE
      ;ENDFOLD
      ;FOLD -- Start Dress in Position AUS -- ;%{SE}%MKUKATPVW %CVW_COM %VCOMMENT %P 2:-- Start Dress in Position AUS --, 3: VW_COMMENT
      ;ENDFOLD
      ;FOLD A3903 = AUS ;%{SE}%MKUKATPVW %CVW_SPS %VBOASG %P 2:A3903 = AUS, 3: BOASG
         $OUT[3903] = FALSE
      ;ENDFOLD
      ;FOLD -- Start Dress Fin AUS -- ;%{SE}%MKUKATPVW %CVW_COM %VCOMMENT %P 2:-- Start Dress Fin AUS --, 3: VW_COMMENT
      ;ENDFOLD
      ;FOLD A3904 = AUS ;%{SE}%MKUKATPVW %CVW_SPS %VBOASG %P 2:A3904 = AUS, 3: BOASG
         $OUT[3904] = FALSE
      ;ENDFOLD
      ;FOLD -- Start StartAcknowledge AUS -- ;%{SE}%MKUKATPVW %CVW_COM %VCOMMENT %P 2:-- Start StartAcknowledge AUS --, 3: VW_COMMENT
      ;ENDFOLD
      ;FOLD A3512 = AUS ;%{SE}%MKUKATPVW %CVW_SPS %VBOASG %P 2:A3512 = AUS, 3: BOASG
         $OUT[3512] = FALSE
      ;ENDFOLD
      ;FOLD -- Schritt Fraesen aktiv -- ;%{SE}%MKUKATPVW %CVW_COM %VCOMMENT %P 2:-- Schritt Fraesen aktiv --, 3: VW_COMMENT
      ;ENDFOLD
      ;FOLD A3534 = AUS ;%{SE}%MKUKATPVW %CVW_SPS %VBOASG %P 2:A3534 = AUS, 3: BOASG
         $OUT[3534] = FALSE
      ;ENDFOLD
      ;FOLD -- Schritt Messen aktiv -- ;%{SE}%MKUKATPVW %CVW_COM %VCOMMENT %P 2:-- Schritt Messen aktiv --, 3: VW_COMMENT
      ;ENDFOLD
      ;FOLD A3535 = AUS ;%{SE}%MKUKATPVW %CVW_SPS %VBOASG %P 2:A3535 = AUS, 3: BOASG
         $OUT[3535] = FALSE
      ;ENDFOLD
      ;FOLD -- Schritt Schweissen aktiv -- ;%{SE}%MKUKATPVW %CVW_COM %VCOMMENT %P 2:-- Schritt Schweissen aktiv --, 3: VW_COMMENT
      ;ENDFOLD
      ;FOLD A3536 = AUS ;%{SE}%MKUKATPVW %CVW_SPS %VBOASG %P 2:A3536 = AUS, 3: BOASG
         $OUT[3536] = FALSE
      ;ENDFOLD
      ;FOLD -- KF1 Ausblasen AUS -- ;%{SE}%MKUKATPVW %CVW_COM %VCOMMENT %P 2:-- KF1 Ausblasen AUS --, 3: VW_COMMENT
      ;ENDFOLD
      ;FOLD A996 = AUS ;%{SE}%MKUKATPVW %CVW_SPS %VBOASG %P 2:A996 = AUS, 3: BOASG
         $OUT[996] = FALSE
      ;ENDFOLD
      ;FOLD -- Ueberwachungszeit ServoGun SZ1 Messen -- ;%{SE}%MKUKATPVW %CVW_COM %VCOMMENT %P 2:-- Ueberwachungszeit ServoGun SZ1 Messen --, 3: VW_COMMENT
      ;ENDFOLD
      ;FOLD t9 ( EIN ) = -150[1/10Sek] ;%{SE}%MKUKATPVW %CVW_SPS %VTASG %P 2:t9 ( EIN ) = -150[1/10Sek], 3: TASG
         VW(#SET_TIME,TRUE,9,0,-150)
      ;ENDFOLD
      ;FOLD -- Fehler SK ruecksetzen -- ;%{SE}%MKUKATPVW %CVW_COM %VCOMMENT %P 2:-- Fehler SK ruecksetzen --, 3: VW_COMMENT
      ;ENDFOLD
      ;FOLD -- Fehler SK Messen AUS -- ;%{SE}%MKUKATPVW %CVW_COM %VCOMMENT %P 2:-- Fehler SK Messen AUS --, 3: VW_COMMENT
      ;ENDFOLD
      ;FOLD F326 = AUS ;%{SE}%MKUKATPVW %CVW_SPS %VBOASG %P 2:F326 = AUS, 3: BOASG
         $FLAG[326] = FALSE
      ;ENDFOLD
      ;FOLD -- Fehler SK Gesamt AUS -- ;%{SE}%MKUKATPVW %CVW_COM %VCOMMENT %P 2:-- Fehler SK Gesamt AUS --, 3: VW_COMMENT
      ;ENDFOLD
      ;FOLD F326 = AUS ;%{SE}%MKUKATPVW %CVW_SPS %VBOASG %P 2:F326 = AUS, 3: BOASG
         $FLAG[326] = FALSE
      ;ENDFOLD
      ;FOLD Schritt 224 = A4039 & A3506 & A3505 & A3894 & !E998 ;%{SE}%MKUKATPVW %CVW_SPS %VST_CON %P 2:Schritt 224 = A4039 & A3506 & A3505 & A3894 & !E998, 3: ST_CON
         IF $OUT[4039] AND $OUT[3506] AND $OUT[3505] AND $OUT[3894] AND NOT $IN[998] THEN
            PREV_STEP[9] = APP_INT_STEP[9]
            APP_INT_STEP[9] = 224
         ENDIF
      ;ENDFOLD
   ;ENDFOLD
   ;FOLD SCHRITT 224 -- st. RZ2 # Init Same -- ;%{P}%MKUKATPVW,%CSTEP,%VST_NR,%P 1:SCHRITT, 2:224, 3: st. RZ2 # Init Same
      ;FOLD ;%{H}
         Case 224
      ;ENDFOLD
      ;FOLD -- Kommentar -- ;%{SE}%MKUKATPVW %CVW_COM %VCOMMENT %P 2:-- Kommentar --, 3: VW_COMMENT
      ;ENDFOLD
      ;FOLD -- Messen nach Fraesen -- ;%{SE}%MKUKATPVW %CVW_COM %VCOMMENT %P 2:-- Messen nach Fraesen --, 3: VW_COMMENT
      ;ENDFOLD
      ;FOLD A3514 = EIN ;%{SE}%MKUKATPVW %CVW_SPS %VBOASG %P 2:A3514 = EIN, 3: BOASG
         $OUT[3514] = TRUE
      ;ENDFOLD
      ;FOLD A3510 = EIN ;%{SE}%MKUKATPVW %CVW_SPS %VBOASG %P 2:A3510 = EIN, 3: BOASG
         $OUT[3510] = TRUE
      ;ENDFOLD
      ;FOLD -- Schritt Messen aktiv -- ;%{SE}%MKUKATPVW %CVW_COM %VCOMMENT %P 2:-- Schritt Messen aktiv --, 3: VW_COMMENT
      ;ENDFOLD
      ;FOLD A3535 = EIN ;%{SE}%MKUKATPVW %CVW_SPS %VBOASG %P 2:A3535 = EIN, 3: BOASG
         $OUT[3535] = TRUE
      ;ENDFOLD
      ;FOLD SCHRITT 225 = A4039 ;%{SE}%MKUKATPVW %CVW_SPS %VST_CON %P 2:SCHRITT 225 = A4039, 3: ST_CON
         IF $OUT[4039] THEN
            PREV_STEP[9] = APP_INT_STEP[9]
            APP_INT_STEP[9] = 225
         ENDIF
      ;ENDFOLD
   ;ENDFOLD
   ;FOLD SCHRITT 225 -- st. RZ2 # Auswertung -- ;%{P}%MKUKATPVW,%CSTEP,%VST_NR,%P 1:SCHRITT, 2:225, 3: st. RZ2 # Auswertung
      ;FOLD ;%{H}
         Case 225
      ;ENDFOLD
      ;FOLD -- Auswertung Messung -- ;%{SE}%MKUKATPVW %CVW_COM %VCOMMENT %P 2:-- Auswertung Messung --, 3: VW_COMMENT
      ;ENDFOLD
      ;FOLD SCHRITT 227 = A4039 & A3508 ;%{SE}%MKUKATPVW %CVW_SPS %VST_CON %P 2:SCHRITT 227 = A4039 & A3508, 3: ST_CON
         IF $OUT[4039] AND $OUT[3508] THEN
            PREV_STEP[9] = APP_INT_STEP[9]
            APP_INT_STEP[9] = 227
         ENDIF
      ;ENDFOLD
      ;FOLD SCHRITT 226 = A4039 & A3509 ;%{SE}%MKUKATPVW %CVW_SPS %VST_CON %P 2:SCHRITT 226 = A4039 & A3509, 3: ST_CON
         IF $OUT[4039] AND $OUT[3509] THEN
            PREV_STEP[9] = APP_INT_STEP[9]
            APP_INT_STEP[9] = 226
         ENDIF
      ;ENDFOLD
   ;ENDFOLD
   ;FOLD SCHRITT 226 -- st. RZ2 # Fehler Messen -- ;%{P}%MKUKATPVW,%CSTEP,%VST_NR,%P 1:SCHRITT, 2:226, 3: st. RZ2 # Fehler Messen
      ;FOLD ;%{H}
         Case 226
      ;ENDFOLD
      ;FOLD -- Start Init Same AUS -- ;%{SE}%MKUKATPVW %CVW_COM %VCOMMENT %P 2:-- Start Init Same AUS --, 3: VW_COMMENT
      ;ENDFOLD
      ;FOLD A3514 = AUS ;%{SE}%MKUKATPVW %CVW_SPS %VBOASG %P 2:A3514 = AUS, 3: BOASG
         $OUT[3514] = FALSE
      ;ENDFOLD
      ;FOLD -- Start Spot AUS -- ;%{SE}%MKUKATPVW %CVW_COM %VCOMMENT %P 2:-- Start Spot AUS --, 3: VW_COMMENT
      ;ENDFOLD
      ;FOLD A3511 = AUS ;%{SE}%MKUKATPVW %CVW_SPS %VBOASG %P 2:A3511 = AUS, 3: BOASG
         $OUT[3511] = FALSE
      ;ENDFOLD
      ;FOLD -- Start Dress AUS -- ;%{SE}%MKUKATPVW %CVW_COM %VCOMMENT %P 2:-- Start Dress AUS --, 3: VW_COMMENT
      ;ENDFOLD
      ;FOLD A3510 = AUS ;%{SE}%MKUKATPVW %CVW_SPS %VBOASG %P 2:A3510 = AUS, 3: BOASG
         $OUT[3510] = FALSE
      ;ENDFOLD
      ;FOLD -- Start Init New AUS -- ;%{SE}%MKUKATPVW %CVW_COM %VCOMMENT %P 2:-- Start Init New AUS --, 3: VW_COMMENT
      ;ENDFOLD
      ;FOLD A3513 = AUS ;%{SE}%MKUKATPVW %CVW_SPS %VBOASG %P 2:A3513 = AUS, 3: BOASG
         $OUT[3513] = FALSE
      ;ENDFOLD
      ;FOLD -- Start Dress in Position AUS -- ;%{SE}%MKUKATPVW %CVW_COM %VCOMMENT %P 2:-- Start Dress in Position AUS --, 3: VW_COMMENT
      ;ENDFOLD
      ;FOLD A3903 = AUS ;%{SE}%MKUKATPVW %CVW_SPS %VBOASG %P 2:A3903 = AUS, 3: BOASG
         $OUT[3903] = FALSE
      ;ENDFOLD
      ;FOLD -- Start Dress Fin AUS -- ;%{SE}%MKUKATPVW %CVW_COM %VCOMMENT %P 2:-- Start Dress Fin AUS --, 3: VW_COMMENT
      ;ENDFOLD
      ;FOLD A3904 = AUS ;%{SE}%MKUKATPVW %CVW_SPS %VBOASG %P 2:A3904 = AUS, 3: BOASG
         $OUT[3904] = FALSE
      ;ENDFOLD
      ;FOLD -- Start StartAcknowledge AUS -- ;%{SE}%MKUKATPVW %CVW_COM %VCOMMENT %P 2:-- Start StartAcknowledge AUS --, 3: VW_COMMENT
      ;ENDFOLD
      ;FOLD A3512 = AUS ;%{SE}%MKUKATPVW %CVW_SPS %VBOASG %P 2:A3512 = AUS, 3: BOASG
         $OUT[3512] = FALSE
      ;ENDFOLD
      ;FOLD -- Kommentar -- ;%{SE}%MKUKATPVW %CVW_COM %VCOMMENT %P 2:-- Kommentar --, 3: VW_COMMENT
      ;ENDFOLD
      ;FOLD -- RSK Sammelstoerung -- ;%{SE}%MKUKATPVW %CVW_COM %VCOMMENT %P 2:-- RSK Sammelstoerung --, 3: VW_COMMENT
      ;ENDFOLD
      ;FOLD F326 = EIN ;%{SE}%MKUKATPVW %CVW_SPS %VBOASG %P 2:F326 = EIN, 3: BOASG
         $FLAG[326] = TRUE
      ;ENDFOLD
      ;FOLD F329 = F326 ;%{SE}%MKUKATPVW %CVW_SPS %VBOASG %P 2:F329 = F326, 3: BOASG
         $FLAG[329] = $FLAG[326]
      ;ENDFOLD
      ;FOLD -- Flagbildung Wiederholfraesen -- ;%{SE}%MKUKATPVW %CVW_COM %VCOMMENT %P 2:-- Flagbildung Wiederholfraesen --, 3: VW_COMMENT
      ;ENDFOLD
      ;FOLD F749 = (F322 + F323 + F325 + F326 + F327 + F329) & !F748 ;%{SE}%MKUKATPVW %CVW_SPS %VBOASG %P 2:F749 = (F322 + F323 + F325 + F326 + F327 + F329) & !F748, 3: BOASG
         $FLAG[749] = ($FLAG[322] OR $FLAG[323] OR $FLAG[325] OR $FLAG[326] OR $FLAG[327] OR $FLAG[329]) AND NOT $FLAG[748]
      ;ENDFOLD
      ;FOLD Schritt 223 = A4039 & F326 & F329 & A3894 & (E26 + E27) ;%{SE}%MKUKATPVW %CVW_SPS %VST_CON %P 2:Schritt 223 = A4039 & F326 & F329 & A3894 & (E26 + E27), 3: ST_CON
         IF $OUT[4039] AND $FLAG[326] AND $FLAG[329] AND $OUT[3894] AND ($IN[26] OR $IN[27]) THEN
            PREV_STEP[9] = APP_INT_STEP[9]
            APP_INT_STEP[9] = 223
         ENDIF
      ;ENDFOLD
      ;FOLD Schritt 250 = A4039 & F326 & F329 & A3894 & A172 ;%{SE}%MKUKATPVW %CVW_SPS %VST_CON %P 2:Schritt 250 = A4039 & F326 & F329 & A3894 & A172, 3: ST_CON
         IF $OUT[4039] AND $FLAG[326] AND $FLAG[329] AND $OUT[3894] AND $OUT[172] THEN
            PREV_STEP[9] = APP_INT_STEP[9]
            APP_INT_STEP[9] = 250
         ENDIF
      ;ENDFOLD
   ;ENDFOLD
   ;FOLD SCHRITT 227 -- st. RZ2 # StartAcknowledge -- ;%{P}%MKUKATPVW,%CSTEP,%VST_NR,%P 1:SCHRITT, 2:227, 3: st. RZ2 # StartAcknowledge
      ;FOLD ;%{H}
         Case 227
      ;ENDFOLD
      ;FOLD -- ServoGun - StartAcknowledge -- ;%{SE}%MKUKATPVW %CVW_COM %VCOMMENT %P 2:-- ServoGun - StartAcknowledge --, 3: VW_COMMENT
      ;ENDFOLD
      ;FOLD -- Start Dress AUS -- ;%{SE}%MKUKATPVW %CVW_COM %VCOMMENT %P 2:-- Start Dress AUS --, 3: VW_COMMENT
      ;ENDFOLD
      ;FOLD A3510 = AUS ;%{SE}%MKUKATPVW %CVW_SPS %VBOASG %P 2:A3510 = AUS, 3: BOASG
         $OUT[3510] = FALSE
      ;ENDFOLD
      ;FOLD -- Start Init Same AUS -- ;%{SE}%MKUKATPVW %CVW_COM %VCOMMENT %P 2:-- Start Init Same AUS --, 3: VW_COMMENT
      ;ENDFOLD
      ;FOLD A3514 = AUS ;%{SE}%MKUKATPVW %CVW_SPS %VBOASG %P 2:A3514 = AUS, 3: BOASG
         $OUT[3514] = FALSE
      ;ENDFOLD
      ;FOLD -- Start StartAcknowledge EIN -- ;%{SE}%MKUKATPVW %CVW_COM %VCOMMENT %P 2:-- Start StartAcknowledge EIN --, 3: VW_COMMENT
      ;ENDFOLD
      ;FOLD A3512 = EIN ;%{SE}%MKUKATPVW %CVW_SPS %VBOASG %P 2:A3512 = EIN, 3: BOASG
         $OUT[3512] = TRUE
      ;ENDFOLD
      ;FOLD -- Schritt Messen aktiv -- ;%{SE}%MKUKATPVW %CVW_COM %VCOMMENT %P 2:-- Schritt Messen aktiv --, 3: VW_COMMENT
      ;ENDFOLD
      ;FOLD A3535 = AUS ;%{SE}%MKUKATPVW %CVW_SPS %VBOASG %P 2:A3535 = AUS, 3: BOASG
         $OUT[3535] = FALSE
      ;ENDFOLD
      ;FOLD SCHRITT 229 = !F335 & A4039 & !A3507 ;%{SE}%MKUKATPVW %CVW_SPS %VST_CON %P 2:SCHRITT 229 = !F335 & A4039 & !A3507, 3: ST_CON
         IF NOT $FLAG[335] AND $OUT[4039] AND NOT $OUT[3507] THEN
            PREV_STEP[9] = APP_INT_STEP[9]
            APP_INT_STEP[9] = 229
         ENDIF
      ;ENDFOLD
      ;FOLD SCHRITT 229 = F335 & !F138 & A4039 & !A3507 ;%{SE}%MKUKATPVW %CVW_SPS %VST_CON %P 2:SCHRITT 229 = F335 & !F138 & A4039 & !A3507, 3: ST_CON
         IF $FLAG[335] AND NOT $FLAG[138] AND $OUT[4039] AND NOT $OUT[3507] THEN
            PREV_STEP[9] = APP_INT_STEP[9]
            APP_INT_STEP[9] = 229
         ENDIF
      ;ENDFOLD
      ;FOLD Schritt 290 = F335 & F138 & A4039 & !A3507 ;%{SE}%MKUKATPVW %CVW_SPS %VST_CON %P 2:Schritt 290 = F335 & F138 & A4039 & !A3507, 3: ST_CON
         IF $FLAG[335] AND $FLAG[138] AND $OUT[4039] AND NOT $OUT[3507] THEN
            PREV_STEP[9] = APP_INT_STEP[9]
            APP_INT_STEP[9] = 290
         ENDIF
      ;ENDFOLD
   ;ENDFOLD
   ;FOLD SCHRITT 229 -- st. RZ2 # Ruecksetzen -- ;%{P}%MKUKATPVW,%CSTEP,%VST_NR,%P 1:SCHRITT, 2:229, 3: st. RZ2 # Ruecksetzen
      ;FOLD ;%{H}
         Case 229
      ;ENDFOLD
      ;FOLD -- Start Init Same AUS -- ;%{SE}%MKUKATPVW %CVW_COM %VCOMMENT %P 2:-- Start Init Same AUS --, 3: VW_COMMENT
      ;ENDFOLD
      ;FOLD A3514 = AUS ;%{SE}%MKUKATPVW %CVW_SPS %VBOASG %P 2:A3514 = AUS, 3: BOASG
         $OUT[3514] = FALSE
      ;ENDFOLD
      ;FOLD -- Start Spot AUS -- ;%{SE}%MKUKATPVW %CVW_COM %VCOMMENT %P 2:-- Start Spot AUS --, 3: VW_COMMENT
      ;ENDFOLD
      ;FOLD A3511 = AUS ;%{SE}%MKUKATPVW %CVW_SPS %VBOASG %P 2:A3511 = AUS, 3: BOASG
         $OUT[3511] = FALSE
      ;ENDFOLD
      ;FOLD -- Start Dress AUS -- ;%{SE}%MKUKATPVW %CVW_COM %VCOMMENT %P 2:-- Start Dress AUS --, 3: VW_COMMENT
      ;ENDFOLD
      ;FOLD A3510 = AUS ;%{SE}%MKUKATPVW %CVW_SPS %VBOASG %P 2:A3510 = AUS, 3: BOASG
         $OUT[3510] = FALSE
      ;ENDFOLD
      ;FOLD -- Start Init New AUS -- ;%{SE}%MKUKATPVW %CVW_COM %VCOMMENT %P 2:-- Start Init New AUS --, 3: VW_COMMENT
      ;ENDFOLD
      ;FOLD A3513 = AUS ;%{SE}%MKUKATPVW %CVW_SPS %VBOASG %P 2:A3513 = AUS, 3: BOASG
         $OUT[3513] = FALSE
      ;ENDFOLD
      ;FOLD -- Start Dress in Position AUS -- ;%{SE}%MKUKATPVW %CVW_COM %VCOMMENT %P 2:-- Start Dress in Position AUS --, 3: VW_COMMENT
      ;ENDFOLD
      ;FOLD A3903 = AUS ;%{SE}%MKUKATPVW %CVW_SPS %VBOASG %P 2:A3903 = AUS, 3: BOASG
         $OUT[3903] = FALSE
      ;ENDFOLD
      ;FOLD -- Start Dress Fin AUS -- ;%{SE}%MKUKATPVW %CVW_COM %VCOMMENT %P 2:-- Start Dress Fin AUS --, 3: VW_COMMENT
      ;ENDFOLD
      ;FOLD A3904 = AUS ;%{SE}%MKUKATPVW %CVW_SPS %VBOASG %P 2:A3904 = AUS, 3: BOASG
         $OUT[3904] = FALSE
      ;ENDFOLD
      ;FOLD -- Start StartAcknowledge AUS -- ;%{SE}%MKUKATPVW %CVW_COM %VCOMMENT %P 2:-- Start StartAcknowledge AUS --, 3: VW_COMMENT
      ;ENDFOLD
      ;FOLD A3512 = AUS ;%{SE}%MKUKATPVW %CVW_SPS %VBOASG %P 2:A3512 = AUS, 3: BOASG
         $OUT[3512] = FALSE
      ;ENDFOLD
      ;FOLD bin30 ( EIN ) = 0 ;%{SE}%MKUKATPVW %CVW_SPS %VARIASG %P 2:bin30 ( EIN ) = 0, 3: ARIASG
         VW(#BINOUT,TRUE,30,0)
      ;ENDFOLD
      ;FOLD -- Schritt Fraesen aktiv -- ;%{SE}%MKUKATPVW %CVW_COM %VCOMMENT %P 2:-- Schritt Fraesen aktiv --, 3: VW_COMMENT
      ;ENDFOLD
      ;FOLD A3534 = AUS ;%{SE}%MKUKATPVW %CVW_SPS %VBOASG %P 2:A3534 = AUS, 3: BOASG
         $OUT[3534] = FALSE
      ;ENDFOLD
      ;FOLD -- Schritt Messen aktiv -- ;%{SE}%MKUKATPVW %CVW_COM %VCOMMENT %P 2:-- Schritt Messen aktiv --, 3: VW_COMMENT
      ;ENDFOLD
      ;FOLD A3535 = AUS ;%{SE}%MKUKATPVW %CVW_SPS %VBOASG %P 2:A3535 = AUS, 3: BOASG
         $OUT[3535] = FALSE
      ;ENDFOLD
      ;FOLD -- Schritt Schweissen aktiv -- ;%{SE}%MKUKATPVW %CVW_COM %VCOMMENT %P 2:-- Schritt Schweissen aktiv --, 3: VW_COMMENT
      ;ENDFOLD
      ;FOLD A3536 = AUS ;%{SE}%MKUKATPVW %CVW_SPS %VBOASG %P 2:A3536 = AUS, 3: BOASG
         $OUT[3536] = FALSE
      ;ENDFOLD
      ;FOLD -- Fehler SK ruecksetzen -- ;%{SE}%MKUKATPVW %CVW_COM %VCOMMENT %P 2:-- Fehler SK ruecksetzen --, 3: VW_COMMENT
      ;ENDFOLD
      ;FOLD -- Druckvorgabe SK1/ServoGun -- ;%{SE}%MKUKATPVW %CVW_COM %VCOMMENT %P 2:-- Druckvorgabe SK1/ServoGun --, 3: VW_COMMENT
      ;ENDFOLD
      ;FOLD bin4 ( F138 ) = 41 ;%{SE}%MKUKATPVW %CVW_SPS %VARIASG %P 2:bin4 ( F138 ) = 41, 3: ARIASG
         VW(#BINOUT,$FLAG[138],4,41)
      ;ENDFOLD
      ;FOLD bin4 ( F139 ) = 51 ;%{SE}%MKUKATPVW %CVW_SPS %VARIASG %P 2:bin4 ( F139 ) = 51, 3: ARIASG
         VW(#BINOUT,$FLAG[139],4,51)
      ;ENDFOLD
      ;FOLD bin31 ( F138 ) = 41 ;%{SE}%MKUKATPVW %CVW_SPS %VARIASG %P 2:bin31 ( F138 ) = 41, 3: ARIASG
         VW(#BINOUT,$FLAG[138],31,41)
      ;ENDFOLD
      ;FOLD bin31 ( F139 ) = 51 ;%{SE}%MKUKATPVW %CVW_SPS %VARIASG %P 2:bin31 ( F139 ) = 51, 3: ARIASG
         VW(#BINOUT,$FLAG[139],31,51)
      ;ENDFOLD
      ;FOLD -- Wartezeit Programmwechsel SK -- ;%{SE}%MKUKATPVW %CVW_COM %VCOMMENT %P 2:-- Wartezeit Programmwechsel SK --, 3: VW_COMMENT
      ;ENDFOLD
      ;FOLD T8 ( !F334 ) = -2[1/10Sek] ;%{SE}%MKUKATPVW %CVW_SPS %VTASG %P 2:T8 ( !F334 ) = -2[1/10Sek], 3: TASG
         VW(#SET_TIME,NOT $FLAG[334],8,0,-2)
      ;ENDFOLD
      ;FOLD -- Hilfsflag SK Programmwechsel -- ;%{SE}%MKUKATPVW %CVW_COM %VCOMMENT %P 2:-- Hilfsflag SK Programmwechsel --, 3: VW_COMMENT
      ;ENDFOLD
      ;FOLD F334 = EIN ;%{SE}%MKUKATPVW %CVW_SPS %VBOASG %P 2:F334 = EIN, 3: BOASG
         $FLAG[334] = TRUE
      ;ENDFOLD
      ;FOLD t9 ( EIN ) = STOP ;%{SE}%MKUKATPVW %CVW_SPS %VTSTOP %P 2:t9 ( EIN ) = STOP, 3: TSTOP
         VW(#SET_TIME,TRUE,9,1,0)
      ;ENDFOLD
      ;FOLD Schritt 230 = T8 & A4039 & A3506 & A3505 & A3894 & !E998 ;%{SE}%MKUKATPVW %CVW_SPS %VST_CON %P 2:Schritt 230 = T8 & A4039 & A3506 & A3505 & A3894 & !E998, 3: ST_CON
         IF $TIMER_FLAG[8] AND $OUT[4039] AND $OUT[3506] AND $OUT[3505] AND $OUT[3894] AND NOT $IN[998] THEN
            PREV_STEP[9] = APP_INT_STEP[9]
            APP_INT_STEP[9] = 230
         ENDIF
      ;ENDFOLD
   ;ENDFOLD
   ;FOLD SCHRITT 230 -- st. RZ2 # Schweissen -- ;%{P}%MKUKATPVW,%CSTEP,%VST_NR,%P 1:SCHRITT, 2:230, 3: st. RZ2 # Schweissen
      ;FOLD ;%{H}
         Case 230
      ;ENDFOLD
      ;FOLD -- Hilfsflag SK Programmwechsel -- ;%{SE}%MKUKATPVW %CVW_COM %VCOMMENT %P 2:-- Hilfsflag SK Programmwechsel --, 3: VW_COMMENT
      ;ENDFOLD
      ;FOLD F334 = AUS ;%{SE}%MKUKATPVW %CVW_SPS %VBOASG %P 2:F334 = AUS, 3: BOASG
         $FLAG[334] = FALSE
      ;ENDFOLD
      ;FOLD A3895 = A3896 & F731 ;%{SE}%MKUKATPVW %CVW_SPS %VBOASG %P 2:A3895 = A3896 & F731, 3: BOASG
         $OUT[3895] = $OUT[3896] AND $FLAG[731]
      ;ENDFOLD
      ;FOLD F748 = A3895 ;%{SE}%MKUKATPVW %CVW_SPS %VBOASG %P 2:F748 = A3895, 3: BOASG
         $FLAG[748] = $OUT[3895]
      ;ENDFOLD
      ;FOLD -- Schritt Schweissen aktiv -- ;%{SE}%MKUKATPVW %CVW_COM %VCOMMENT %P 2:-- Schritt Schweissen aktiv --, 3: VW_COMMENT
      ;ENDFOLD
      ;FOLD A3536 = EIN ;%{SE}%MKUKATPVW %CVW_SPS %VBOASG %P 2:A3536 = EIN, 3: BOASG
         $OUT[3536] = TRUE
      ;ENDFOLD
      ;FOLD -- ServoGun - Start Spot EIN -- ;%{SE}%MKUKATPVW %CVW_COM %VCOMMENT %P 2:-- ServoGun - Start Spot EIN --, 3: VW_COMMENT
      ;ENDFOLD
      ;FOLD A3511 = EIN ;%{SE}%MKUKATPVW %CVW_SPS %VBOASG %P 2:A3511 = EIN, 3: BOASG
         $OUT[3511] = TRUE
      ;ENDFOLD
      ;FOLD F749 = AUS ;%{SE}%MKUKATPVW %CVW_SPS %VBOASG %P 2:F749 = AUS, 3: BOASG
         $FLAG[749] = FALSE
      ;ENDFOLD
      ;FOLD SCHRITT 231 = A4039 ;%{SE}%MKUKATPVW %CVW_SPS %VST_CON %P 2:SCHRITT 231 = A4039, 3: ST_CON
         IF $OUT[4039] THEN
            PREV_STEP[9] = APP_INT_STEP[9]
            APP_INT_STEP[9] = 231
         ENDIF
      ;ENDFOLD
   ;ENDFOLD
   ;FOLD SCHRITT 231 -- st. RZ2 # Auswertung -- ;%{P}%MKUKATPVW,%CSTEP,%VST_NR,%P 1:SCHRITT, 2:231, 3: st. RZ2 # Auswertung
      ;FOLD ;%{H}
         Case 231
      ;ENDFOLD
      ;FOLD -- Auswertung -- ;%{SE}%MKUKATPVW %CVW_COM %VCOMMENT %P 2:-- Auswertung --, 3: VW_COMMENT
      ;ENDFOLD
      ;FOLD Schritt 232 = A3509 & !E964 & E965 ;%{SE}%MKUKATPVW %CVW_SPS %VST_CON %P 2:Schritt 232 = A3509 & !E964 & E965, 3: ST_CON
         IF $OUT[3509] AND NOT $IN[964] AND $IN[965] THEN
            PREV_STEP[9] = APP_INT_STEP[9]
            APP_INT_STEP[9] = 232
         ENDIF
      ;ENDFOLD
      ;FOLD SCHRITT 233 = A3508 & (E964 & !E966 + !A945 & E15) ;%{SE}%MKUKATPVW %CVW_SPS %VST_CON %P 2:SCHRITT 233 = A3508 & (E964 & !E966 + !A945 & E15), 3: ST_CON
         IF $OUT[3508] AND ($IN[964] AND NOT $IN[966] OR NOT $OUT[945] AND $IN[15]) THEN
            PREV_STEP[9] = APP_INT_STEP[9]
            APP_INT_STEP[9] = 233
         ENDIF
      ;ENDFOLD
   ;ENDFOLD
   ;FOLD SCHRITT 232 -- st. RZ2 # Fehler Schweissung -- ;%{P}%MKUKATPVW,%CSTEP,%VST_NR,%P 1:SCHRITT, 2:232, 3: st. RZ2 # Fehler Schweissung
      ;FOLD ;%{H}
         Case 232
      ;ENDFOLD
      ;FOLD -- Start Init Same AUS -- ;%{SE}%MKUKATPVW %CVW_COM %VCOMMENT %P 2:-- Start Init Same AUS --, 3: VW_COMMENT
      ;ENDFOLD
      ;FOLD A3514 = AUS ;%{SE}%MKUKATPVW %CVW_SPS %VBOASG %P 2:A3514 = AUS, 3: BOASG
         $OUT[3514] = FALSE
      ;ENDFOLD
      ;FOLD -- Start Spot AUS -- ;%{SE}%MKUKATPVW %CVW_COM %VCOMMENT %P 2:-- Start Spot AUS --, 3: VW_COMMENT
      ;ENDFOLD
      ;FOLD A3511 = AUS ;%{SE}%MKUKATPVW %CVW_SPS %VBOASG %P 2:A3511 = AUS, 3: BOASG
         $OUT[3511] = FALSE
      ;ENDFOLD
      ;FOLD -- Start Dress AUS -- ;%{SE}%MKUKATPVW %CVW_COM %VCOMMENT %P 2:-- Start Dress AUS --, 3: VW_COMMENT
      ;ENDFOLD
      ;FOLD A3510 = AUS ;%{SE}%MKUKATPVW %CVW_SPS %VBOASG %P 2:A3510 = AUS, 3: BOASG
         $OUT[3510] = FALSE
      ;ENDFOLD
      ;FOLD -- Start Init New AUS -- ;%{SE}%MKUKATPVW %CVW_COM %VCOMMENT %P 2:-- Start Init New AUS --, 3: VW_COMMENT
      ;ENDFOLD
      ;FOLD A3513 = AUS ;%{SE}%MKUKATPVW %CVW_SPS %VBOASG %P 2:A3513 = AUS, 3: BOASG
         $OUT[3513] = FALSE
      ;ENDFOLD
      ;FOLD -- Start Dress in Position AUS -- ;%{SE}%MKUKATPVW %CVW_COM %VCOMMENT %P 2:-- Start Dress in Position AUS --, 3: VW_COMMENT
      ;ENDFOLD
      ;FOLD A3903 = AUS ;%{SE}%MKUKATPVW %CVW_SPS %VBOASG %P 2:A3903 = AUS, 3: BOASG
         $OUT[3903] = FALSE
      ;ENDFOLD
      ;FOLD -- Start Dress Fin AUS -- ;%{SE}%MKUKATPVW %CVW_COM %VCOMMENT %P 2:-- Start Dress Fin AUS --, 3: VW_COMMENT
      ;ENDFOLD
      ;FOLD A3904 = AUS ;%{SE}%MKUKATPVW %CVW_SPS %VBOASG %P 2:A3904 = AUS, 3: BOASG
         $OUT[3904] = FALSE
      ;ENDFOLD
      ;FOLD -- Start StartAcknowledge AUS -- ;%{SE}%MKUKATPVW %CVW_COM %VCOMMENT %P 2:-- Start StartAcknowledge AUS --, 3: VW_COMMENT
      ;ENDFOLD
      ;FOLD A3512 = AUS ;%{SE}%MKUKATPVW %CVW_SPS %VBOASG %P 2:A3512 = AUS, 3: BOASG
         $OUT[3512] = FALSE
      ;ENDFOLD
      ;FOLD -- RSK Fehlerausgabe Kraftaufbau -- ;%{SE}%MKUKATPVW %CVW_COM %VCOMMENT %P 2:-- RSK Fehlerausgabe Kraftaufbau --, 3: VW_COMMENT
      ;ENDFOLD
      ;FOLD F325 = EIN ;%{SE}%MKUKATPVW %CVW_SPS %VBOASG %P 2:F325 = EIN, 3: BOASG
         $FLAG[325] = TRUE
      ;ENDFOLD
      ;FOLD -- RSK Fehlerausgabe -- ;%{SE}%MKUKATPVW %CVW_COM %VCOMMENT %P 2:-- RSK Fehlerausgabe --, 3: VW_COMMENT
      ;ENDFOLD
      ;FOLD F327 = EIN ;%{SE}%MKUKATPVW %CVW_SPS %VBOASG %P 2:F327 = EIN, 3: BOASG
         $FLAG[327] = TRUE
      ;ENDFOLD
      ;FOLD F138 = !F327 & F138 ;%{SE}%MKUKATPVW %CVW_SPS %VBOASG %P 2:F138 = !F327 & F138, 3: BOASG
         $FLAG[138] = NOT $FLAG[327] AND $FLAG[138]
      ;ENDFOLD
      ;FOLD F139 = F327 + F139 ;%{SE}%MKUKATPVW %CVW_SPS %VBOASG %P 2:F139 = F327 + F139, 3: BOASG
         $FLAG[139] = $FLAG[327] OR $FLAG[139]
      ;ENDFOLD
      ;FOLD -- RSK Sammelstoerung -- ;%{SE}%MKUKATPVW %CVW_COM %VCOMMENT %P 2:-- RSK Sammelstoerung --, 3: VW_COMMENT
      ;ENDFOLD
      ;FOLD F329 = F325 + F326 + F327 ;%{SE}%MKUKATPVW %CVW_SPS %VBOASG %P 2:F329 = F325 + F326 + F327, 3: BOASG
         $FLAG[329] = $FLAG[325] OR $FLAG[326] OR $FLAG[327]
      ;ENDFOLD
      ;FOLD A3519 = EIN ;%{SE}%MKUKATPVW %CVW_SPS %VBOASG %P 2:A3519 = EIN, 3: BOASG
         $OUT[3519] = TRUE
      ;ENDFOLD
      ;FOLD -- Flagbildung Wiederholfraesen -- ;%{SE}%MKUKATPVW %CVW_COM %VCOMMENT %P 2:-- Flagbildung Wiederholfraesen --, 3: VW_COMMENT
      ;ENDFOLD
      ;FOLD F749 = F329 & !A3518 ;%{SE}%MKUKATPVW %CVW_SPS %VBOASG %P 2:F749 = F329 & !A3518, 3: BOASG
         $FLAG[749] = $FLAG[329] AND NOT $OUT[3518]
      ;ENDFOLD
      ;FOLD A176 = A3518 ;%{SE}%MKUKATPVW %CVW_SPS %VBOASG %P 2:A176 = A3518, 3: BOASG
         $OUT[176] = $OUT[3518]
      ;ENDFOLD
      ;FOLD Schritt 265 = A3894 & A3518 ;%{SE}%MKUKATPVW %CVW_SPS %VST_CON %P 2:Schritt 265 = A3894 & A3518, 3: ST_CON
         IF $OUT[3894] AND $OUT[3518] THEN
            PREV_STEP[9] = APP_INT_STEP[9]
            APP_INT_STEP[9] = 265
         ENDIF
      ;ENDFOLD
      ;FOLD Schritt 203 = A3894 & !A3518 & F749 & A4039 ;%{SE}%MKUKATPVW %CVW_SPS %VST_CON %P 2:Schritt 203 = A3894 & !A3518 & F749 & A4039, 3: ST_CON
         IF $OUT[3894] AND NOT $OUT[3518] AND $FLAG[749] AND $OUT[4039] THEN
            PREV_STEP[9] = APP_INT_STEP[9]
            APP_INT_STEP[9] = 203
         ENDIF
      ;ENDFOLD
   ;ENDFOLD
   ;FOLD SCHRITT 233 -- st. RZ2 # StartAcknowledge -- ;%{P}%MKUKATPVW,%CSTEP,%VST_NR,%P 1:SCHRITT, 2:233, 3: st. RZ2 # StartAcknowledge
      ;FOLD ;%{H}
         Case 233
